LIN {X 0,Y 192.833,Z 984.62,A -85,B 0,C 180,E1 9990.303,E2 9990.303} C_VEL
LIN {X 0,Y 192.693,Z 984.368,A -85,B 0,C 180,E1 9985.841,E2 9985.841} C_VEL
LIN {X 0,Y 192.486,Z 982.897,A -85,B 0,C 180,E1 9980.438,E2 9980.438} C_VEL
LIN {X 0,Y 192.915,Z 979.845,A -85,B 0,C 180,E1 9974.58,E2 9974.58} C_VEL
LIN {X 0,Y 194.824,Z 974.779,A -85,B 0,C 180,E1 9968.005,E2 9968.005} C_VEL
LIN {X 0,Y 198.477,Z 968.183,A -85,B 0,C 180,E1 9961.744,E2 9961.744} C_VEL
LIN {X 0,Y 204.063,Z 959.66,A -85,B 0,C 180,E1 9955.712,E2 9955.712} C_VEL
LIN {X 0,Y 211.597,Z 949.246,A -85,B 0,C 180,E1 9950.02,E2 9950.02} C_VEL
LIN {X 0,Y 220.496,Z 937.345,A -85,B 0,C 180,E1 9944.986,E2 9944.986} C_VEL
LIN {X 0,Y 230.256,Z 924.203,A -85,B 0,C 180,E1 9940.643,E2 9940.643} C_VEL
LIN {X 0,Y 240.936,Z 909.167,A -85,B 0,C 180,E1 9936.792,E2 9936.792} C_VEL
LIN {X 0,Y 251.155,Z 893.767,A -85,B 0,C 180,E1 9933.703,E2 9933.703} C_VEL
LIN {X 0,Y 261.767,Z 876.537,A -85,B 0,C 180,E1 9930.974,E2 9930.974} C_VEL
LIN {X 0,Y 271.504,Z 859.077,A -85,B 0,C 180,E1 9928.793,E2 9928.793} C_VEL
LIN {X 0,Y 280.905,Z 840.055,A -85,B 0,C 180,E1 9926.934,E2 9926.934} C_VEL
LIN {X 0,Y 289.057,Z 821.044,A -85,B 0,C 180,E1 9925.484,E2 9925.484} C_VEL
LIN {X 0,Y 296.643,Z 800.32,A -85,B 0,C 180,E1 9924.267,E2 9924.267} C_VEL
LIN {X 0,Y 302.941,Z 779.468,A -85,B 0,C 180,E1 9923.354,E2 9923.354} C_VEL
LIN {X 0,Y 308.032,Z 757.203,A -85,B 0,C 180,E1 9922.636,E2 9922.636} C_VEL
LIN {X 0,Y 311.388,Z 735.251,A -85,B 0,C 180,E1 9922.089,E2 9922.089} C_VEL
LIN {X 0,Y 327.083,Z 591.178,A -85,B 0,C 180,E1 9919.092,E2 9919.092} C_VEL
LIN {X 0,Y 325.532,Z 586.958,A -85,B 0,C 180,E1 9917.057,E2 9917.057} C_VEL
LIN {X 0,Y 324.558,Z 584.437,A -85,B 0,C 180,E1 9915.363,E2 9915.363} C_VEL
LIN {X 0,Y 323.649,Z 581.615,A -85,B 0,C 180,E1 9912.307,E2 9912.307} C_VEL
LIN {X 0,Y 323.587,Z 581.778,A -85,B 0,C 180,E1 9909.425,E2 9909.425} C_VEL
LIN {X 0,Y 324.621,Z 585.303,A -85,B 0,C 180,E1 9906.011,E2 9906.011} C_VEL
LIN {X 0,Y 326.028,Z 589.355,A -85,B 0,C 180,E1 9903.692,E2 9903.692} C_VEL
LIN {X 0,Y 326.424,Z 590.965,A -85,B 0,C 180,E1 9903.104,E2 9903.104} C_VEL
LIN {X 0,Y 309.523,Z 735.661,A -85,B 0,C 180,E1 9900.051,E2 9900.051} C_VEL
LIN {X 0,Y 305.578,Z 756.66,A -85,B 0,C 180,E1 9899.378,E2 9899.378} C_VEL
LIN {X 0,Y 300.528,Z 776.512,A -85,B 0,C 180,E1 9898.509,E2 9898.509} C_VEL
LIN {X 0,Y 294.236,Z 796.168,A -85,B 0,C 180,E1 9897.379,E2 9897.379} C_VEL
LIN {X 0,Y 287.043,Z 814.874,A -85,B 0,C 180,E1 9896.005,E2 9896.005} C_VEL
LIN {X 0,Y 278.796,Z 832.848,A -85,B 0,C 180,E1 9894.326,E2 9894.326} C_VEL
LIN {X 0,Y 269.408,Z 850.655,A -85,B 0,C 180,E1 9892.227,E2 9892.227} C_VEL
LIN {X 0,Y 259.717,Z 866.928,A -85,B 0,C 180,E1 9889.799,E2 9889.799} C_VEL
LIN {X 0,Y 250.062,Z 881.523,A -85,B 0,C 180,E1 9887.06,E2 9887.06} C_VEL
LIN {X 0,Y 239.647,Z 895.837,A -85,B 0,C 180,E1 9883.636,E2 9883.636} C_VEL
LIN {X 0,Y 229.516,Z 908.579,A -85,B 0,C 180,E1 9879.684,E2 9879.684} C_VEL
LIN {X 0,Y 220.368,Z 919.385,A -85,B 0,C 180,E1 9875.327,E2 9875.327} C_VEL
LIN {X 0,Y 211.892,Z 928.983,A -85,B 0,C 180,E1 9870.24,E2 9870.24} C_VEL
LIN {X 0,Y 205.09,Z 936.539,A -85,B 0,C 180,E1 9864.88,E2 9864.88} C_VEL
LIN {X 0,Y 199.749,Z 942.543,A -85,B 0,C 180,E1 9859.024,E2 9859.024} C_VEL
LIN {X 0,Y 196,Z 946.905,A -85,B 0,C 180,E1 9852.714,E2 9852.714} C_VEL
LIN {X 0,Y 194.012,Z 949.301,A -85,B 0,C 180,E1 9846.704,E2 9846.704} C_VEL
LIN {X 0,Y 193.164,Z 950.247,A -85,B 0,C 180,E1 9840.766,E2 9840.766} C_VEL
LIN {X 0,Y 193.005,Z 949.923,A -85,B 0,C 180,E1 9835.458,E2 9835.458} C_VEL
LIN {X 0,Y 193.369,Z 948.241,A -85,B 0,C 180,E1 9829.765,E2 9829.765} C_VEL
LIN {X 0,Y 194.609,Z 945.069,A -85,B 0,C 180,E1 9823.819,E2 9823.819} C_VEL
LIN {X 0,Y 197.11,Z 940.246,A -85,B 0,C 180,E1 9817.865,E2 9817.865} C_VEL
LIN {X 0,Y 201.137,Z 933.501,A -85,B 0,C 180,E1 9811.988,E2 9811.988} C_VEL
LIN {X 0,Y 206.391,Z 925.353,A -85,B 0,C 180,E1 9806.661,E2 9806.661} C_VEL
LIN {X 0,Y 213.003,Z 915.362,A -85,B 0,C 180,E1 9801.627,E2 9801.627} C_VEL
LIN {X 0,Y 220.514,Z 903.893,A -85,B 0,C 180,E1 9797.129,E2 9797.129} C_VEL
LIN {X 0,Y 228.48,Z 891.228,A -85,B 0,C 180,E1 9793.207,E2 9793.207} C_VEL
LIN {X 0,Y 237.374,Z 876.099,A -85,B 0,C 180,E1 9789.532,E2 9789.532} C_VEL
LIN {X 0,Y 245.848,Z 860.287,A -85,B 0,C 180,E1 9786.507,E2 9786.507} C_VEL
LIN {X 0,Y 253.94,Z 843.552,A -85,B 0,C 180,E1 9783.954,E2 9783.954} C_VEL
LIN {X 0,Y 261.811,Z 825.226,A -85,B 0,C 180,E1 9781.73,E2 9781.73} C_VEL
LIN {X 0,Y 268.975,Z 805.916,A -85,B 0,C 180,E1 9779.874,E2 9779.874} C_VEL
LIN {X 0,Y 274.986,Z 786.777,A -85,B 0,C 180,E1 9778.423,E2 9778.423} C_VEL
LIN {X 0,Y 280.418,Z 765.377,A -85,B 0,C 180,E1 9777.178,E2 9777.178} C_VEL
LIN {X 0,Y 284.657,Z 743.254,A -85,B 0,C 180,E1 9776.242,E2 9776.242} C_VEL
LIN {X 0,Y 287.486,Z 721.546,A -85,B 0,C 180,E1 9775.613,E2 9775.613} C_VEL
LIN {X 0,Y 300.678,Z 576.179,A -85,B 0,C 180,E1 9772.398,E2 9772.398} C_VEL
LIN {X 0,Y 293.024,Z 562.174,A -85,B 0,C 180,E1 9768.58,E2 9768.58} C_VEL
LIN {X 0,Y 286.481,Z 551.351,A -85,B 0,C 180,E1 9764.831,E2 9764.831} C_VEL
LIN {X 0,Y 281.715,Z 543.744,A -85,B 0,C 180,E1 9761.651,E2 9761.651} C_VEL
LIN {X 0,Y 278.454,Z 538.921,A -85,B 0,C 180,E1 9759.197,E2 9759.197} C_VEL
LIN {X 0,Y 275.745,Z 534.842,A -85,B 0,C 180,E1 9756.878,E2 9756.878} C_VEL
LIN {X 0,Y 272.521,Z 530.083,A -85,B 0,C 180,E1 9753.643,E2 9753.643} C_VEL
LIN {X 0,Y 269.339,Z 525.473,A -85,B 0,C 180,E1 9749.587,E2 9749.587} C_VEL
LIN {X 0,Y 266.095,Z 520.826,A -85,B 0,C 180,E1 9742.98,E2 9742.98} C_VEL
LIN {X 0,Y 265.114,Z 519.942,A -85,B 0,C 180,E1 9737.561,E2 9737.561} C_VEL
LIN {X 0,Y 265.642,Z 520.425,A -85,B 0,C 180,E1 9732.389,E2 9732.389} C_VEL
LIN {X 0,Y 266.487,Z 521.324,A -85,B 0,C 180,E1 9729.721,E2 9729.721} C_VEL
LIN {X 0,Y 267.942,Z 523.757,A -85,B 0,C 180,E1 9726.466,E2 9726.466} C_VEL
LIN {X 0,Y 268.633,Z 525.593,A -85,B 0,C 180,E1 9725.108,E2 9725.108} C_VEL
LIN {X 0,Y 269.61,Z 530.896,A -85,B 0,C 180,E1 9723.019,E2 9723.019} C_VEL
LIN {X 0,Y 270.981,Z 536.847,A -85,B 0,C 180,E1 9720.737,E2 9720.737} C_VEL
LIN {X 0,Y 271.921,Z 538.54,A -85,B 0,C 180,E1 9719.631,E2 9719.631} C_VEL
LIN {X 0,Y 276.165,Z 545.02,A -85,B 0,C 180,E1 9715.536,E2 9715.536} C_VEL
LIN {X 0,Y 280.055,Z 550.846,A -85,B 0,C 180,E1 9712.461,E2 9712.461} C_VEL
LIN {X 0,Y 284.859,Z 558.419,A -85,B 0,C 180,E1 9709.177,E2 9709.177} C_VEL
LIN {X 0,Y 291.313,Z 568.942,A -85,B 0,C 180,E1 9705.389,E2 9705.389} C_VEL
LIN {X 0,Y 298.171,Z 581.104,A -85,B 0,C 180,E1 9701.88,E2 9701.88} C_VEL
LIN {X 0,Y 300.746,Z 586.097,A -85,B 0,C 180,E1 9700.666,E2 9700.666} C_VEL
LIN {X 0,Y 286.5,Z 747.246,A -85,B 0,C 180,E1 9697.213,E2 9697.213} C_VEL
LIN {X 0,Y 282.924,Z 769.359,A -85,B 0,C 180,E1 9696.541,E2 9696.541} C_VEL
LIN {X 0,Y 278.126,Z 790.293,A -85,B 0,C 180,E1 9695.696,E2 9695.696} C_VEL
LIN {X 0,Y 272.318,Z 810.598,A -85,B 0,C 180,E1 9694.592,E2 9694.592} C_VEL
LIN {X 0,Y 265.286,Z 830.997,A -85,B 0,C 180,E1 9693.136,E2 9693.136} C_VEL
LIN {X 0,Y 257.466,Z 850.135,A -85,B 0,C 180,E1 9691.368,E2 9691.368} C_VEL
LIN {X 0,Y 249.024,Z 868.363,A -85,B 0,C 180,E1 9689.237,E2 9689.237} C_VEL
LIN {X 0,Y 240.302,Z 885.289,A -85,B 0,C 180,E1 9686.761,E2 9686.761} C_VEL
LIN {X 0,Y 230.867,Z 901.925,A -85,B 0,C 180,E1 9683.669,E2 9683.669} C_VEL
LIN {X 0,Y 221.57,Z 917.018,A -85,B 0,C 180,E1 9680.105,E2 9680.105} C_VEL
LIN {X 0,Y 212.413,Z 931.213,A -85,B 0,C 180,E1 9675.842,E2 9675.842} C_VEL
LIN {X 0,Y 204.126,Z 943.761,A -85,B 0,C 180,E1 9671.03,E2 9671.03} C_VEL
LIN {X 0,Y 197.069,Z 954.627,A -85,B 0,C 180,E1 9665.701,E2 9665.701} C_VEL
LIN {X 0,Y 191.38,Z 963.9,A -85,B 0,C 180,E1 9659.763,E2 9659.763} C_VEL
LIN {X 0,Y 187.435,Z 971.453,A -85,B 0,C 180,E1 9653.436,E2 9653.436} C_VEL
LIN {X 0,Y 185.25,Z 977.221,A -85,B 0,C 180,E1 9646.951,E2 9646.951} C_VEL
LIN {X 0,Y 184.584,Z 980.952,A -85,B 0,C 180,E1 9640.935,E2 9640.935} C_VEL
LIN {X 0,Y 184.709,Z 983.16,A -85,B 0,C 180,E1 9635.123,E2 9635.123} C_VEL
LIN {X 0,Y 184.866,Z 983.888,A -85,B 0,C 180,E1 9630.316,E2 9630.316} C_VEL
LIN {X 0,Y 184.729,Z 983.696,A -85,B 0,C 180,E1 9625.972,E2 9625.972} C_VEL
LIN {X 0,Y 184.506,Z 982.433,A -85,B 0,C 180,E1 9620.651,E2 9620.651} C_VEL
LIN {X 0,Y 184.977,Z 979.342,A -85,B 0,C 180,E1 9614.182,E2 9614.182} C_VEL
LIN {X 0,Y 187.036,Z 974.447,A -85,B 0,C 180,E1 9607.37,E2 9607.37} C_VEL
LIN {X 0,Y 190.947,Z 967.93,A -85,B 0,C 180,E1 9600.866,E2 9600.866} C_VEL
LIN {X 0,Y 196.888,Z 959.58,A -85,B 0,C 180,E1 9594.634,E2 9594.634} C_VEL
LIN {X 0,Y 205.273,Z 948.796,A -85,B 0,C 180,E1 9588.523,E2 9588.523} C_VEL
LIN {X 0,Y 214.698,Z 936.999,A -85,B 0,C 180,E1 9583.417,E2 9583.417} C_VEL
LIN {X 0,Y 225.087,Z 923.789,A -85,B 0,C 180,E1 9578.991,E2 9578.991} C_VEL
LIN {X 0,Y 235.457,Z 909.867,A -85,B 0,C 180,E1 9575.393,E2 9575.393} C_VEL
LIN {X 0,Y 246.713,Z 893.8,A -85,B 0,C 180,E1 9572.123,E2 9572.123} C_VEL
LIN {X 0,Y 257.323,Z 877.334,A -85,B 0,C 180,E1 9569.51,E2 9569.51} C_VEL
LIN {X 0,Y 267.72,Z 859.507,A -85,B 0,C 180,E1 9567.283,E2 9567.283} C_VEL
LIN {X 0,Y 277.372,Z 840.653,A -85,B 0,C 180,E1 9565.46,E2 9565.46} C_VEL
LIN {X 0,Y 286.134,Z 821.067,A -85,B 0,C 180,E1 9563.982,E2 9563.982} C_VEL
LIN {X 0,Y 293.67,Z 801.296,A -85,B 0,C 180,E1 9562.838,E2 9562.838} C_VEL
LIN {X 0,Y 300.384,Z 779.833,A -85,B 0,C 180,E1 9561.914,E2 9561.914} C_VEL
LIN {X 0,Y 305.639,Z 757.703,A -85,B 0,C 180,E1 9561.213,E2 9561.213} C_VEL
LIN {X 0,Y 309.183,Z 735.886,A -85,B 0,C 180,E1 9560.674,E2 9560.674} C_VEL
LIN {X 0,Y 324.902,Z 596.612,A -85,B 0,C 180,E1 9557.784,E2 9557.784} C_VEL
LIN {X 0,Y 323.461,Z 592.436,A -85,B 0,C 180,E1 9555.348,E2 9555.348} C_VEL
LIN {X 0,Y 322.547,Z 589.523,A -85,B 0,C 180,E1 9552.168,E2 9552.168} C_VEL
LIN {X 0,Y 322.489,Z 589.614,A -85,B 0,C 180,E1 9549.638,E2 9549.638} C_VEL
LIN {X 0,Y 323.363,Z 593.042,A -85,B 0,C 180,E1 9546.301,E2 9546.301} C_VEL
LIN {X 0,Y 324.38,Z 596.39,A -85,B 0,C 180,E1 9544.389,E2 9544.389} C_VEL
LIN {X 0,Y 307.554,Z 736.129,A -85,B 0,C 180,E1 9541.49,E2 9541.49} C_VEL
LIN {X 0,Y 303.512,Z 757.009,A -85,B 0,C 180,E1 9540.838,E2 9540.838} C_VEL
LIN {X 0,Y 298.202,Z 777.251,A -85,B 0,C 180,E1 9539.971,E2 9539.971} C_VEL
LIN {X 0,Y 291.469,Z 797.614,A -85,B 0,C 180,E1 9538.82,E2 9538.82} C_VEL
LIN {X 0,Y 284.2,Z 815.824,A -85,B 0,C 180,E1 9537.501,E2 9537.501} C_VEL
LIN {X 0,Y 275.605,Z 833.879,A -85,B 0,C 180,E1 9535.838,E2 9535.838} C_VEL
LIN {X 0,Y 266.445,Z 850.698,A -85,B 0,C 180,E1 9533.892,E2 9533.892} C_VEL
LIN {X 0,Y 256.248,Z 867.217,A -85,B 0,C 180,E1 9531.472,E2 9531.472} C_VEL
LIN {X 0,Y 246.173,Z 881.917,A -85,B 0,C 180,E1 9528.757,E2 9528.757} C_VEL
LIN {X 0,Y 235.124,Z 896.392,A -85,B 0,C 180,E1 9525.31,E2 9525.31} C_VEL
LIN {X 0,Y 225.137,Z 908.385,A -85,B 0,C 180,E1 9521.619,E2 9521.619} C_VEL
LIN {X 0,Y 215.144,Z 919.598,A -85,B 0,C 180,E1 9517.132,E2 9517.132} C_VEL
LIN {X 0,Y 206.072,Z 929.273,A -85,B 0,C 180,E1 9511.998,E2 9511.998} C_VEL
LIN {X 0,Y 198.479,Z 937.134,A -85,B 0,C 180,E1 9506.348,E2 9506.348} C_VEL
LIN {X 0,Y 192.659,Z 943.167,A -85,B 0,C 180,E1 9500.33,E2 9500.33} C_VEL
LIN {X 0,Y 188.407,Z 947.646,A -85,B 0,C 180,E1 9493.611,E2 9493.611} C_VEL
LIN {X 0,Y 186.19,Z 950.04,A -85,B 0,C 180,E1 9487.35,E2 9487.35} C_VEL
LIN {X 0,Y 185.228,Z 950.979,A -85,B 0,C 180,E1 9481.203,E2 9481.203} C_VEL
LIN {X 0,Y 185.035,Z 950.641,A -85,B 0,C 180,E1 9475.522,E2 9475.522} C_VEL
LIN {X 0,Y 185.385,Z 949.048,A -85,B 0,C 180,E1 9469.856,E2 9469.856} C_VEL
LIN {X 0,Y 186.585,Z 946.14,A -85,B 0,C 180,E1 9463.947,E2 9463.947} C_VEL
LIN {X 0,Y 189.209,Z 941.259,A -85,B 0,C 180,E1 9457.585,E2 9457.585} C_VEL
LIN {X 0,Y 193.152,Z 934.985,A -85,B 0,C 180,E1 9451.773,E2 9451.773} C_VEL
LIN {X 0,Y 198.874,Z 926.59,A -85,B 0,C 180,E1 9445.958,E2 9445.958} C_VEL
LIN {X 0,Y 205.756,Z 916.723,A -85,B 0,C 180,E1 9440.766,E2 9440.766} C_VEL
LIN {X 0,Y 213.506,Z 905.467,A -85,B 0,C 180,E1 9436.177,E2 9436.177} C_VEL
LIN {X 0,Y 222.324,Z 892.027,A -85,B 0,C 180,E1 9431.917,E2 9431.917} C_VEL
LIN {X 0,Y 231.494,Z 877.004,A -85,B 0,C 180,E1 9428.222,E2 9428.222} C_VEL
LIN {X 0,Y 240.341,Z 861.098,A -85,B 0,C 180,E1 9425.15,E2 9425.15} C_VEL
LIN {X 0,Y 248.705,Z 844.401,A -85,B 0,C 180,E1 9422.588,E2 9422.588} C_VEL
LIN {X 0,Y 256.822,Z 826.129,A -85,B 0,C 180,E1 9420.363,E2 9420.363} C_VEL
LIN {X 0,Y 263.861,Z 807.884,A -85,B 0,C 180,E1 9418.594,E2 9418.594} C_VEL
LIN {X 0,Y 270.378,Z 787.882,A -85,B 0,C 180,E1 9417.066,E2 9417.066} C_VEL
LIN {X 0,Y 275.951,Z 766.589,A -85,B 0,C 180,E1 9415.828,E2 9415.828} C_VEL
LIN {X 0,Y 280.233,Z 745.122,A -85,B 0,C 180,E1 9414.912,E2 9414.912} C_VEL
LIN {X 0,Y 283.214,Z 723.651,A -85,B 0,C 180,E1 9414.275,E2 9414.275} C_VEL
LIN {X 0,Y 296.636,Z 580.476,A -85,B 0,C 180,E1 9411.135,E2 9411.135} C_VEL
LIN {X 0,Y 289.758,Z 567.709,A -85,B 0,C 180,E1 9407.519,E2 9407.519} C_VEL
LIN {X 0,Y 283.334,Z 556.902,A -85,B 0,C 180,E1 9403.623,E2 9403.623} C_VEL
LIN {X 0,Y 278.597,Z 549.234,A -85,B 0,C 180,E1 9400.242,E2 9400.242} C_VEL
LIN {X 0,Y 274.037,Z 542.29,A -85,B 0,C 180,E1 9396.364,E2 9396.364} C_VEL
LIN {X 0,Y 271.016,Z 537.705,A -85,B 0,C 180,E1 9393.221,E2 9393.221} C_VEL
LIN {X 0,Y 267.959,Z 533.166,A -85,B 0,C 180,E1 9389.168,E2 9389.168} C_VEL
LIN {X 0,Y 264.982,Z 528.733,A -85,B 0,C 180,E1 9382.871,E2 9382.871} C_VEL
LIN {X 0,Y 264.034,Z 527.866,A -85,B 0,C 180,E1 9377.381,E2 9377.381} C_VEL
LIN {X 0,Y 264.615,Z 528.399,A -85,B 0,C 180,E1 9372.217,E2 9372.217} C_VEL
LIN {X 0,Y 265.391,Z 529.314,A -85,B 0,C 180,E1 9369.762,E2 9369.762} C_VEL
LIN {X 0,Y 268.904,Z 534.267,A -85,B 0,C 180,E1 9363.305,E2 9363.305} C_VEL
LIN {X 0,Y 271.921,Z 538.54,A -85,B 0,C 180,E1 9359.631,E2 9359.631} C_VEL
LIN {X 0,Y 273.084,Z 540.822,A -85,B 0,C 180,E1 9358.351,E2 9358.351} C_VEL
LIN {X 0,Y 274.504,Z 546.424,A -85,B 0,C 180,E1 9356.636,E2 9356.636} C_VEL
LIN {X 0,Y 276.478,Z 554.666,A -85,B 0,C 180,E1 9354.425,E2 9354.425} C_VEL
LIN {X 0,Y 277.625,Z 557.294,A -85,B 0,C 180,E1 9353.422,E2 9353.422} C_VEL
LIN {X 0,Y 282.668,Z 565.44,A -85,B 0,C 180,E1 9349.814,E2 9349.814} C_VEL
LIN {X 0,Y 288.966,Z 575.986,A -85,B 0,C 180,E1 9345.984,E2 9345.984} C_VEL
LIN {X 0,Y 295.773,Z 588.381,A -85,B 0,C 180,E1 9342.389,E2 9342.389} C_VEL
LIN {X 0,Y 296.668,Z 590.18,A -85,B 0,C 180,E1 9341.944,E2 9341.944} C_VEL
LIN {X 0,Y 282.411,Z 747.03,A -85,B 0,C 180,E1 9338.602,E2 9338.602} C_VEL
LIN {X 0,Y 278.737,Z 769.213,A -85,B 0,C 180,E1 9337.934,E2 9337.934} C_VEL
LIN {X 0,Y 273.812,Z 790.175,A -85,B 0,C 180,E1 9337.098,E2 9337.098} C_VEL
LIN {X 0,Y 267.699,Z 810.918,A -85,B 0,C 180,E1 9335.977,E2 9335.977} C_VEL
LIN {X 0,Y 260.565,Z 831.016,A -85,B 0,C 180,E1 9334.547,E2 9334.547} C_VEL
LIN {X 0,Y 252.454,Z 850.268,A -85,B 0,C 180,E1 9332.773,E2 9332.773} C_VEL
LIN {X 0,Y 243.777,Z 868.376,A -85,B 0,C 180,E1 9330.649,E2 9330.649} C_VEL
LIN {X 0,Y 234.454,Z 885.785,A -85,B 0,C 180,E1 9328.073,E2 9328.073} C_VEL
LIN {X 0,Y 224.73,Z 902.341,A -85,B 0,C 180,E1 9324.956,E2 9324.956} C_VEL
LIN {X 0,Y 215.12,Z 917.318,A -85,B 0,C 180,E1 9321.345,E2 9321.345} C_VEL
LIN {X 0,Y 205.926,Z 930.916,A -85,B 0,C 180,E1 9317.159,E2 9317.159} C_VEL
LIN {X 0,Y 197.333,Z 943.293,A -85,B 0,C 180,E1 9312.29,E2 9312.29} C_VEL
LIN {X 0,Y 189.965,Z 954.037,A -85,B 0,C 180,E1 9306.868,E2 9306.868} C_VEL
LIN {X 0,Y 183.925,Z 963.302,A -85,B 0,C 180,E1 9300.737,E2 9300.737} C_VEL
LIN {X 0,Y 179.77,Z 970.689,A -85,B 0,C 180,E1 9294.311,E2 9294.311} C_VEL
LIN {X 0,Y 177.417,Z 976.359,A -85,B 0,C 180,E1 9287.724,E2 9287.724} C_VEL
LIN {X 0,Y 176.622,Z 980.126,A -85,B 0,C 180,E1 9281.435,E2 9281.435} C_VEL
LIN {X 0,Y 176.731,Z 982.41,A -85,B 0,C 180,E1 9275.312,E2 9275.312} C_VEL
LIN {X 0,Y 176.899,Z 983.157,A -85,B 0,C 180,E1 9270.331,E2 9270.331} C_VEL
LIN {X 0,Y 176.746,Z 982.982,A -85,B 0,C 180,E1 9265.79,E2 9265.79} C_VEL
LIN {X 0,Y 176.522,Z 981.732,A -85,B 0,C 180,E1 9260.224,E2 9260.224} C_VEL
LIN {X 0,Y 177.069,Z 978.772,A -85,B 0,C 180,E1 9253.608,E2 9253.608} C_VEL
LIN {X 0,Y 179.27,Z 974.121,A -85,B 0,C 180,E1 9246.68,E2 9246.68} C_VEL
LIN {X 0,Y 183.465,Z 967.693,A -85,B 0,C 180,E1 9239.917,E2 9239.917} C_VEL
LIN {X 0,Y 189.789,Z 959.502,A -85,B 0,C 180,E1 9233.474,E2 9233.474} C_VEL
LIN {X 0,Y 198.199,Z 949.467,A -85,B 0,C 180,E1 9227.479,E2 9227.479} C_VEL
LIN {X 0,Y 208.007,Z 937.998,A -85,B 0,C 180,E1 9222.258,E2 9222.258} C_VEL
LIN {X 0,Y 218.763,Z 924.999,A -85,B 0,C 180,E1 9217.761,E2 9217.761} C_VEL
LIN {X 0,Y 230.132,Z 910.653,A -85,B 0,C 180,E1 9213.93,E2 9213.93} C_VEL
LIN {X 0,Y 242.116,Z 894.38,A -85,B 0,C 180,E1 9210.58,E2 9210.58} C_VEL
LIN {X 0,Y 253.061,Z 878.242,A -85,B 0,C 180,E1 9208,E2 9208} C_VEL
LIN {X 0,Y 264.552,Z 859.227,A -85,B 0,C 180,E1 9205.652,E2 9205.652} C_VEL
LIN {X 0,Y 274.44,Z 840.62,A -85,B 0,C 180,E1 9203.886,E2 9203.886} C_VEL
LIN {X 0,Y 283.832,Z 820.224,A -85,B 0,C 180,E1 9202.391,E2 9202.391} C_VEL
LIN {X 0,Y 291.786,Z 799.829,A -85,B 0,C 180,E1 9201.258,E2 9201.258} C_VEL
LIN {X 0,Y 298.408,Z 779.132,A -85,B 0,C 180,E1 9200.407,E2 9200.407} C_VEL
LIN {X 0,Y 303.791,Z 756.859,A -85,B 0,C 180,E1 9199.728,E2 9199.728} C_VEL
LIN {X 0,Y 307.441,Z 734.943,A -85,B 0,C 180,E1 9199.203,E2 9199.203} C_VEL
LIN {X 0,Y 322.953,Z 602.452,A -85,B 0,C 180,E1 9196.502,E2 9196.502} C_VEL
LIN {X 0,Y 322.097,Z 599.9,A -85,B 0,C 180,E1 9194.746,E2 9194.746} C_VEL
LIN {X 0,Y 321.441,Z 597.431,A -85,B 0,C 180,E1 9192.028,E2 9192.028} C_VEL
LIN {X 0,Y 321.388,Z 597.633,A -85,B 0,C 180,E1 9189.671,E2 9189.671} C_VEL
LIN {X 0,Y 322.111,Z 600.78,A -85,B 0,C 180,E1 9186.595,E2 9186.595} C_VEL
LIN {X 0,Y 322.487,Z 602.369,A -85,B 0,C 180,E1 9185.68,E2 9185.68} C_VEL
LIN {X 0,Y 305.848,Z 736.59,A -85,B 0,C 180,E1 9182.949,E2 9182.949} C_VEL
LIN {X 0,Y 301.647,Z 757.664,A -85,B 0,C 180,E1 9182.308,E2 9182.308} C_VEL
LIN {X 0,Y 296.367,Z 777.386,A -85,B 0,C 180,E1 9181.49,E2 9181.49} C_VEL
LIN {X 0,Y 289.582,Z 797.446,A -85,B 0,C 180,E1 9180.395,E2 9180.395} C_VEL
LIN {X 0,Y 281.646,Z 816.695,A -85,B 0,C 180,E1 9179.036,E2 9179.036} C_VEL
LIN {X 0,Y 272.714,Z 834.906,A -85,B 0,C 180,E1 9177.395,E2 9177.395} C_VEL
LIN {X 0,Y 262.923,Z 852.151,A -85,B 0,C 180,E1 9175.419,E2 9175.419} C_VEL
LIN {X 0,Y 251.862,Z 869.301,A -85,B 0,C 180,E1 9172.908,E2 9172.908} C_VEL
LIN {X 0,Y 241.026,Z 884.238,A -85,B 0,C 180,E1 9170.1,E2 9170.1} C_VEL
LIN {X 0,Y 230.033,Z 897.994,A -85,B 0,C 180,E1 9166.784,E2 9166.784} C_VEL
LIN {X 0,Y 219.142,Z 910.356,A -85,B 0,C 180,E1 9162.89,E2 9162.89} C_VEL
LIN {X 0,Y 209.337,Z 920.709,A -85,B 0,C 180,E1 9158.631,E2 9158.631} C_VEL
LIN {X 0,Y 199.919,Z 930.11,A -85,B 0,C 180,E1 9153.521,E2 9153.521} C_VEL
LIN {X 0,Y 192.016,Z 937.749,A -85,B 0,C 180,E1 9147.917,E2 9147.917} C_VEL
LIN {X 0,Y 185.674,Z 943.797,A -85,B 0,C 180,E1 9141.736,E2 9141.736} C_VEL
LIN {X 0,Y 181.057,Z 948.186,A -85,B 0,C 180,E1 9134.969,E2 9134.969} C_VEL
LIN {X 0,Y 178.469,Z 950.7,A -85,B 0,C 180,E1 9128.339,E2 9128.339} C_VEL
LIN {X 0,Y 177.299,Z 951.716,A -85,B 0,C 180,E1 9121.618,E2 9121.618} C_VEL
LIN {X 0,Y 177.063,Z 951.379,A -85,B 0,C 180,E1 9115.765,E2 9115.765} C_VEL
LIN {X 0,Y 177.424,Z 949.776,A -85,B 0,C 180,E1 9109.755,E2 9109.755} C_VEL
LIN {X 0,Y 178.698,Z 946.872,A -85,B 0,C 180,E1 9103.584,E2 9103.584} C_VEL
LIN {X 0,Y 181.493,Z 941.99,A -85,B 0,C 180,E1 9096.954,E2 9096.954} C_VEL
LIN {X 0,Y 185.678,Z 935.723,A -85,B 0,C 180,E1 9090.919,E2 9090.919} C_VEL
LIN {X 0,Y 191.734,Z 927.322,A -85,B 0,C 180,E1 9084.902,E2 9084.902} C_VEL
LIN {X 0,Y 198.967,Z 917.472,A -85,B 0,C 180,E1 9079.571,E2 9079.571} C_VEL
LIN {X 0,Y 207.085,Z 906.228,A -85,B 0,C 180,E1 9074.881,E2 9074.881} C_VEL
LIN {X 0,Y 216.285,Z 892.799,A -85,B 0,C 180,E1 9070.553,E2 9070.553} C_VEL
LIN {X 0,Y 225.292,Z 878.607,A -85,B 0,C 180,E1 9067.006,E2 9067.006} C_VEL
LIN {X 0,Y 234.35,Z 863.02,A -85,B 0,C 180,E1 9063.926,E2 9063.926} C_VEL
LIN {X 0,Y 243.288,Z 845.903,A -85,B 0,C 180,E1 9061.255,E2 9061.255} C_VEL
LIN {X 0,Y 251.64,Z 827.8,A -85,B 0,C 180,E1 9059.028,E2 9059.028} C_VEL
LIN {X 0,Y 258.877,Z 809.786,A -85,B 0,C 180,E1 9057.263,E2 9057.263} C_VEL
LIN {X 0,Y 265.541,Z 790.017,A -85,B 0,C 180,E1 9055.744,E2 9055.744} C_VEL
LIN {X 0,Y 271.09,Z 769.788,A -85,B 0,C 180,E1 9054.546,E2 9054.546} C_VEL
LIN {X 0,Y 275.682,Z 748.23,A -85,B 0,C 180,E1 9053.594,E2 9053.594} C_VEL
LIN {X 0,Y 279.065,Z 725.551,A -85,B 0,C 180,E1 9052.9,E2 9052.9} C_VEL
LIN {X 0,Y 292.657,Z 584.756,A -85,B 0,C 180,E1 9049.823,E2 9049.823} C_VEL
LIN {X 0,Y 286.599,Z 573.391,A -85,B 0,C 180,E1 9046.451,E2 9046.451} C_VEL
LIN {X 0,Y 280.78,Z 563.239,A -85,B 0,C 180,E1 9042.717,E2 9042.717} C_VEL
LIN {X 0,Y 275.847,Z 555.059,A -85,B 0,C 180,E1 9038.968,E2 9038.968} C_VEL
LIN {X 0,Y 272.238,Z 549.579,A -85,B 0,C 180,E1 9035.731,E2 9035.731} C_VEL
LIN {X 0,Y 269.525,Z 545.326,A -85,B 0,C 180,E1 9032.795,E2 9032.795} C_VEL
LIN {X 0,Y 266.706,Z 540.984,A -85,B 0,C 180,E1 9028.922,E2 9028.922} C_VEL
LIN {X 0,Y 263.793,Z 536.569,A -85,B 0,C 180,E1 9022.509,E2 9022.509} C_VEL
LIN {X 0,Y 262.951,Z 535.78,A -85,B 0,C 180,E1 9017.026,E2 9017.026} C_VEL
LIN {X 0,Y 263.655,Z 536.42,A -85,B 0,C 180,E1 9011.818,E2 9011.818} C_VEL
LIN {X 0,Y 264.294,Z 537.302,A -85,B 0,C 180,E1 9009.802,E2 9009.802} C_VEL
LIN {X 0,Y 267.64,Z 542.148,A -85,B 0,C 180,E1 9003.535,E2 9003.535} C_VEL
LIN {X 0,Y 271.021,Z 547.224,A -85,B 0,C 180,E1 8999.366,E2 8999.366} C_VEL
LIN {X 0,Y 274.451,Z 552.464,A -85,B 0,C 180,E1 8996.031,E2 8996.031} C_VEL
LIN {X 0,Y 277.625,Z 557.294,A -85,B 0,C 180,E1 8993.422,E2 8993.422} C_VEL
LIN {X 0,Y 279.241,Z 561.173,A -85,B 0,C 180,E1 8992.082,E2 8992.082} C_VEL
LIN {X 0,Y 281.518,Z 570.097,A -85,B 0,C 180,E1 8990.083,E2 8990.083} C_VEL
LIN {X 0,Y 283.661,Z 577.43,A -85,B 0,C 180,E1 8988.408,E2 8988.408} C_VEL
LIN {X 0,Y 284.501,Z 579.252,A -85,B 0,C 180,E1 8987.863,E2 8987.863} C_VEL
LIN {X 0,Y 290.309,Z 589.84,A -85,B 0,C 180,E1 8984.52,E2 8984.52} C_VEL
LIN {X 0,Y 292.711,Z 594.573,A -85,B 0,C 180,E1 8983.25,E2 8983.25} C_VEL
LIN {X 0,Y 278.461,Z 746.627,A -85,B 0,C 180,E1 8980.03,E2 8980.03} C_VEL
LIN {X 0,Y 274.717,Z 768.754,A -85,B 0,C 180,E1 8979.371,E2 8979.371} C_VEL
LIN {X 0,Y 269.664,Z 789.808,A -85,B 0,C 180,E1 8978.545,E2 8978.545} C_VEL
LIN {X 0,Y 263.186,Z 811.189,A -85,B 0,C 180,E1 8977.402,E2 8977.402} C_VEL
LIN {X 0,Y 256.072,Z 830.722,A -85,B 0,C 180,E1 8976.026,E2 8976.026} C_VEL
LIN {X 0,Y 247.599,Z 850.33,A -85,B 0,C 180,E1 8974.235,E2 8974.235} C_VEL
LIN {X 0,Y 238.683,Z 868.367,A -85,B 0,C 180,E1 8972.123,E2 8972.123} C_VEL
LIN {X 0,Y 228.735,Z 886.28,A -85,B 0,C 180,E1 8969.452,E2 8969.452} C_VEL
LIN {X 0,Y 219.331,Z 901.723,A -85,B 0,C 180,E1 8966.524,E2 8966.524} C_VEL
LIN {X 0,Y 209.371,Z 916.662,A -85,B 0,C 180,E1 8962.901,E2 8962.901} C_VEL
LIN {X 0,Y 199.69,Z 930.383,A -85,B 0,C 180,E1 8958.63,E2 8958.63} C_VEL
LIN {X 0,Y 190.384,Z 943.158,A -85,B 0,C 180,E1 8953.478,E2 8953.478} C_VEL
LIN {X 0,Y 182.87,Z 953.537,A -85,B 0,C 180,E1 8948.065,E2 8948.065} C_VEL
LIN {X 0,Y 176.526,Z 962.679,A -85,B 0,C 180,E1 8941.794,E2 8941.794} C_VEL
LIN {X 0,Y 172.066,Z 970.053,A -85,B 0,C 180,E1 8935.107,E2 8935.107} C_VEL
LIN {X 0,Y 169.524,Z 975.708,A -85,B 0,C 180,E1 8928.223,E2 8928.223} C_VEL
LIN {X 0,Y 168.648,Z 979.466,A -85,B 0,C 180,E1 8921.636,E2 8921.636} C_VEL
LIN {X 0,Y 168.757,Z 981.672,A -85,B 0,C 180,E1 8915.447,E2 8915.447} C_VEL
LIN {X 0,Y 168.932,Z 982.423,A -85,B 0,C 180,E1 8910.346,E2 8910.346} C_VEL
LIN {X 0,Y 168.763,Z 982.27,A -85,B 0,C 180,E1 8905.59,E2 8905.59} C_VEL
LIN {X 0,Y 168.543,Z 981.099,A -85,B 0,C 180,E1 8899.983,E2 8899.983} C_VEL
LIN {X 0,Y 169.212,Z 978.119,A -85,B 0,C 180,E1 8892.824,E2 8892.824} C_VEL
LIN {X 0,Y 171.694,Z 973.524,A -85,B 0,C 180,E1 8885.586,E2 8885.586} C_VEL
LIN {X 0,Y 176.584,Z 966.792,A -85,B 0,C 180,E1 8878.234,E2 8878.234} C_VEL
LIN {X 0,Y 183.535,Z 958.594,A -85,B 0,C 180,E1 8871.617,E2 8871.617} C_VEL
LIN {X 0,Y 192.615,Z 948.54,A -85,B 0,C 180,E1 8865.521,E2 8865.521} C_VEL
LIN {X 0,Y 203.07,Z 937.065,A -85,B 0,C 180,E1 8860.266,E2 8860.266} C_VEL
LIN {X 0,Y 214.435,Z 924.102,A -85,B 0,C 180,E1 8855.787,E2 8855.787} C_VEL
LIN {X 0,Y 226.338,Z 909.753,A -85,B 0,C 180,E1 8852,E2 8852} C_VEL
LIN {X 0,Y 238.437,Z 894.022,A -85,B 0,C 180,E1 8848.801,E2 8848.801} C_VEL
LIN {X 0,Y 249.945,Z 877.707,A -85,B 0,C 180,E1 8846.237,E2 8846.237} C_VEL
LIN {X 0,Y 261.116,Z 859.855,A -85,B 0,C 180,E1 8844.075,E2 8844.075} C_VEL
LIN {X 0,Y 271.314,Z 841.483,A -85,B 0,C 180,E1 8842.349,E2 8842.349} C_VEL
LIN {X 0,Y 280.918,Z 821.522,A -85,B 0,C 180,E1 8840.901,E2 8840.901} C_VEL
LIN {X 0,Y 289.035,Z 801.68,A -85,B 0,C 180,E1 8839.809,E2 8839.809} C_VEL
LIN {X 0,Y 295.99,Z 780.791,A -85,B 0,C 180,E1 8838.96,E2 8838.96} C_VEL
LIN {X 0,Y 301.537,Z 759.265,A -85,B 0,C 180,E1 8838.309,E2 8838.309} C_VEL
LIN {X 0,Y 305.682,Z 736.194,A -85,B 0,C 180,E1 8837.759,E2 8837.759} C_VEL
LIN {X 0,Y 321.172,Z 608.612,A -85,B 0,C 180,E1 8835.208,E2 8835.208} C_VEL
LIN {X 0,Y 320.337,Z 605.339,A -85,B 0,C 180,E1 8831.888,E2 8831.888} C_VEL
LIN {X 0,Y 320.29,Z 605.469,A -85,B 0,C 180,E1 8829.886,E2 8829.886} C_VEL
LIN {X 0,Y 320.833,Z 608.382,A -85,B 0,C 180,E1 8826.986,E2 8826.986} C_VEL
LIN {X 0,Y 304.394,Z 737.285,A -85,B 0,C 180,E1 8824.42,E2 8824.42} C_VEL
LIN {X 0,Y 300.107,Z 758.295,A -85,B 0,C 180,E1 8823.8,E2 8823.8} C_VEL
LIN {X 0,Y 294.606,Z 778.207,A -85,B 0,C 180,E1 8822.998,E2 8822.998} C_VEL
LIN {X 0,Y 287.593,Z 798.265,A -85,B 0,C 180,E1 8821.932,E2 8821.932} C_VEL
LIN {X 0,Y 279.456,Z 817.462,A -85,B 0,C 180,E1 8820.614,E2 8820.614} C_VEL
LIN {X 0,Y 270.468,Z 835.208,A -85,B 0,C 180,E1 8819.059,E2 8819.059} C_VEL
LIN {X 0,Y 260.264,Z 852.648,A -85,B 0,C 180,E1 8817.114,E2 8817.114} C_VEL
LIN {X 0,Y 248.992,Z 869.552,A -85,B 0,C 180,E1 8814.7,E2 8814.7} C_VEL
LIN {X 0,Y 238.071,Z 884.128,A -85,B 0,C 180,E1 8812.033,E2 8812.033} C_VEL
LIN {X 0,Y 226.325,Z 898.23,A -85,B 0,C 180,E1 8808.703,E2 8808.703} C_VEL
LIN {X 0,Y 214.537,Z 911.015,A -85,B 0,C 180,E1 8804.71,E2 8804.71} C_VEL
LIN {X 0,Y 203.649,Z 921.87,A -85,B 0,C 180,E1 8800.197,E2 8800.197} C_VEL
LIN {X 0,Y 193.597,Z 931.287,A -85,B 0,C 180,E1 8794.943,E2 8794.943} C_VEL
LIN {X 0,Y 185.111,Z 938.88,A -85,B 0,C 180,E1 8789.126,E2 8789.126} C_VEL
LIN {X 0,Y 178.353,Z 944.821,A -85,B 0,C 180,E1 8782.737,E2 8782.737} C_VEL
LIN {X 0,Y 173.373,Z 949.161,A -85,B 0,C 180,E1 8775.641,E2 8775.641} C_VEL
LIN {X 0,Y 170.612,Z 951.54,A -85,B 0,C 180,E1 8768.789,E2 8768.789} C_VEL
LIN {X 0,Y 169.337,Z 952.456,A -85,B 0,C 180,E1 8761.693,E2 8761.693} C_VEL
LIN {X 0,Y 169.098,Z 952.065,A -85,B 0,C 180,E1 8755.563,E2 8755.563} C_VEL
LIN {X 0,Y 169.512,Z 950.367,A -85,B 0,C 180,E1 8749.279,E2 8749.279} C_VEL
LIN {X 0,Y 171.035,Z 947.153,A -85,B 0,C 180,E1 8742.484,E2 8742.484} C_VEL
LIN {X 0,Y 174.199,Z 942.156,A -85,B 0,C 180,E1 8735.592,E2 8735.592} C_VEL
LIN {X 0,Y 179.102,Z 935.352,A -85,B 0,C 180,E1 8729.034,E2 8729.034} C_VEL
LIN {X 0,Y 185.382,Z 927.124,A -85,B 0,C 180,E1 8723.179,E2 8723.179} C_VEL
LIN {X 0,Y 193.154,Z 917.044,A -85,B 0,C 180,E1 8717.74,E2 8717.74} C_VEL
LIN {X 0,Y 201.816,Z 905.507,A -85,B 0,C 180,E1 8712.979,E2 8712.979} C_VEL
LIN {X 0,Y 210.931,Z 892.698,A -85,B 0,C 180,E1 8708.879,E2 8708.879} C_VEL
LIN {X 0,Y 220.337,Z 878.408,A -85,B 0,C 180,E1 8705.319,E2 8705.319} C_VEL
LIN {X 0,Y 229.753,Z 862.643,A -85,B 0,C 180,E1 8702.243,E2 8702.243} C_VEL
LIN {X 0,Y 238.509,Z 846.318,A -85,B 0,C 180,E1 8699.722,E2 8699.722} C_VEL
LIN {X 0,Y 247.291,Z 827.786,A -85,B 0,C 180,E1 8697.465,E2 8697.465} C_VEL
LIN {X 0,Y 254.867,Z 809.292,A -85,B 0,C 180,E1 8695.686,E2 8695.686} C_VEL
LIN {X 0,Y 261.61,Z 789.74,A -85,B 0,C 180,E1 8694.21,E2 8694.21} C_VEL
LIN {X 0,Y 267.211,Z 769.663,A -85,B 0,C 180,E1 8693.047,E2 8693.047} C_VEL
LIN {X 0,Y 271.844,Z 748.301,A -85,B 0,C 180,E1 8692.122,E2 8692.122} C_VEL
LIN {X 0,Y 275.282,Z 725.694,A -85,B 0,C 180,E1 8691.442,E2 8691.442} C_VEL
LIN {X 0,Y 288.808,Z 589.059,A -85,B 0,C 180,E1 8688.475,E2 8688.475} C_VEL
LIN {X 0,Y 283.775,Z 579.461,A -85,B 0,C 180,E1 8685.506,E2 8685.506} C_VEL
LIN {X 0,Y 278.038,Z 569.141,A -85,B 0,C 180,E1 8681.623,E2 8681.623} C_VEL
LIN {X 0,Y 273.401,Z 561.555,A -85,B 0,C 180,E1 8677.909,E2 8677.909} C_VEL
LIN {X 0,Y 270.571,Z 557.02,A -85,B 0,C 180,E1 8675.204,E2 8675.204} C_VEL
LIN {X 0,Y 268.049,Z 552.946,A -85,B 0,C 180,E1 8672.363,E2 8672.363} C_VEL
LIN {X 0,Y 265.403,Z 548.74,A -85,B 0,C 180,E1 8668.585,E2 8668.585} C_VEL
LIN {X 0,Y 262.663,Z 544.456,A -85,B 0,C 180,E1 8662.322,E2 8662.322} C_VEL
LIN {X 0,Y 261.877,Z 543.702,A -85,B 0,C 180,E1 8656.869,E2 8656.869} C_VEL
LIN {X 0,Y 262.707,Z 544.447,A -85,B 0,C 180,E1 8651.415,E2 8651.415} C_VEL
LIN {X 0,Y 263.787,Z 546.473,A -85,B 0,C 180,E1 8648.282,E2 8648.282} C_VEL
LIN {X 0,Y 266.306,Z 549.883,A -85,B 0,C 180,E1 8643.876,E2 8643.876} C_VEL
LIN {X 0,Y 269.516,Z 554.832,A -85,B 0,C 180,E1 8639.788,E2 8639.788} C_VEL
LIN {X 0,Y 272.864,Z 560.1,A -85,B 0,C 180,E1 8636.429,E2 8636.429} C_VEL
LIN {X 0,Y 276.79,Z 566.26,A -85,B 0,C 180,E1 8633.154,E2 8633.154} C_VEL
LIN {X 0,Y 281.961,Z 574.853,A -85,B 0,C 180,E1 8629.478,E2 8629.478} C_VEL
LIN {X 0,Y 284.501,Z 579.252,A -85,B 0,C 180,E1 8627.863,E2 8627.863} C_VEL
LIN {X 0,Y 285.595,Z 582.684,A -85,B 0,C 180,E1 8627.105,E2 8627.105} C_VEL
LIN {X 0,Y 287.436,Z 595.248,A -85,B 0,C 180,E1 8625.427,E2 8625.427} C_VEL
LIN {X 0,Y 288.315,Z 597.695,A -85,B 0,C 180,E1 8624.887,E2 8624.887} C_VEL
LIN {X 0,Y 288.831,Z 599.021,A -85,B 0,C 180,E1 8624.583,E2 8624.583} C_VEL
LIN {X 0,Y 274.676,Z 746.227,A -85,B 0,C 180,E1 8621.496,E2 8621.496} C_VEL
LIN {X 0,Y 270.847,Z 768.418,A -85,B 0,C 180,E1 8620.845,E2 8620.845} C_VEL
LIN {X 0,Y 265.693,Z 789.434,A -85,B 0,C 180,E1 8620.037,E2 8620.037} C_VEL
LIN {X 0,Y 259.052,Z 810.849,A -85,B 0,C 180,E1 8618.912,E2 8618.912} C_VEL
LIN {X 0,Y 251.591,Z 830.76,A -85,B 0,C 180,E1 8617.525,E2 8617.525} C_VEL
LIN {X 0,Y 242.908,Z 850.307,A -85,B 0,C 180,E1 8615.755,E2 8615.755} C_VEL
LIN {X 0,Y 233.752,Z 868.252,A -85,B 0,C 180,E1 8613.661,E2 8613.661} C_VEL
LIN {X 0,Y 223.667,Z 885.845,A -85,B 0,C 180,E1 8611.046,E2 8611.046} C_VEL
LIN {X 0,Y 213.486,Z 901.961,A -85,B 0,C 180,E1 8607.971,E2 8607.971} C_VEL
LIN {X 0,Y 203.164,Z 916.894,A -85,B 0,C 180,E1 8604.303,E2 8604.303} C_VEL
LIN {X 0,Y 193.191,Z 930.369,A -85,B 0,C 180,E1 8600.001,E2 8600.001} C_VEL
LIN {X 0,Y 183.42,Z 943.114,A -85,B 0,C 180,E1 8594.692,E2 8594.692} C_VEL
LIN {X 0,Y 175.271,Z 953.747,A -85,B 0,C 180,E1 8588.874,E2 8588.874} C_VEL
LIN {X 0,Y 168.617,Z 962.909,A -85,B 0,C 180,E1 8582.262,E2 8582.262} C_VEL
LIN {X 0,Y 164.034,Z 970.061,A -85,B 0,C 180,E1 8575.265,E2 8575.265} C_VEL
LIN {X 0,Y 161.386,Z 975.715,A -85,B 0,C 180,E1 8567.68,E2 8567.68} C_VEL
LIN {X 0,Y 160.639,Z 979.297,A -85,B 0,C 180,E1 8560.769,E2 8560.769} C_VEL
LIN {X 0,Y 160.818,Z 981.109,A -85,B 0,C 180,E1 8554.643,E2 8554.643} C_VEL
LIN {X 0,Y 160.962,Z 981.714,A -85,B 0,C 180,E1 8549.652,E2 8549.652} C_VEL
LIN {X 0,Y 160.748,Z 981.473,A -85,B 0,C 180,E1 8544.654,E2 8544.654} C_VEL
LIN {X 0,Y 160.598,Z 980.054,A -85,B 0,C 180,E1 8538.152,E2 8538.152} C_VEL
LIN {X 0,Y 161.758,Z 976.72,A -85,B 0,C 180,E1 8530.51,E2 8530.51} C_VEL
LIN {X 0,Y 165.392,Z 971.238,A -85,B 0,C 180,E1 8522.267,E2 8522.267} C_VEL
LIN {X 0,Y 171.138,Z 964.518,A -85,B 0,C 180,E1 8515.081,E2 8515.081} C_VEL
LIN {X 0,Y 179.624,Z 955.533,A -85,B 0,C 180,E1 8508.1,E2 8508.1} C_VEL
LIN {X 0,Y 189.896,Z 944.945,A -85,B 0,C 180,E1 8502.075,E2 8502.075} C_VEL
LIN {X 0,Y 201.428,Z 932.921,A -85,B 0,C 180,E1 8496.961,E2 8496.961} C_VEL
LIN {X 0,Y 213.733,Z 919.486,A -85,B 0,C 180,E1 8492.656,E2 8492.656} C_VEL
LIN {X 0,Y 226.438,Z 904.617,A -85,B 0,C 180,E1 8489.053,E2 8489.053} C_VEL
LIN {X 0,Y 238.838,Z 888.684,A -85,B 0,C 180,E1 8486.123,E2 8486.123} C_VEL
LIN {X 0,Y 250.618,Z 871.935,A -85,B 0,C 180,E1 8483.762,E2 8483.762} C_VEL
LIN {X 0,Y 262.119,Z 853.601,A -85,B 0,C 180,E1 8481.763,E2 8481.763} C_VEL
LIN {X 0,Y 272.219,Z 835.307,A -85,B 0,C 180,E1 8480.225,E2 8480.225} C_VEL
LIN {X 0,Y 281.238,Z 816.178,A -85,B 0,C 180,E1 8478.989,E2 8478.989} C_VEL
LIN {X 0,Y 289.112,Z 796.389,A -85,B 0,C 180,E1 8478.02,E2 8478.02} C_VEL
LIN {X 0,Y 296.112,Z 774.815,A -85,B 0,C 180,E1 8477.242,E2 8477.242} C_VEL
LIN {X 0,Y 301.498,Z 752.99,A -85,B 0,C 180,E1 8476.644,E2 8476.644} C_VEL
LIN {X 0,Y 305.263,Z 730.155,A -85,B 0,C 180,E1 8476.146,E2 8476.146} C_VEL
LIN {X 0,Y 319.593,Z 615.147,A -85,B 0,C 180,E1 8473.893,E2 8473.893} C_VEL
LIN {X 0,Y 319.235,Z 613.248,A -85,B 0,C 180,E1 8471.746,E2 8471.746} C_VEL
LIN {X 0,Y 319.189,Z 613.486,A -85,B 0,C 180,E1 8469.92,E2 8469.92} C_VEL
LIN {X 0,Y 319.342,Z 615.128,A -85,B 0,C 180,E1 8468.294,E2 8468.294} C_VEL
LIN {X 0,Y 303.282,Z 737.768,A -85,B 0,C 180,E1 8465.913,E2 8465.913} C_VEL
LIN {X 0,Y 298.867,Z 758.826,A -85,B 0,C 180,E1 8465.313,E2 8465.313} C_VEL
LIN {X 0,Y 293.355,Z 778.295,A -85,B 0,C 180,E1 8464.558,E2 8464.558} C_VEL
LIN {X 0,Y 285.963,Z 798.972,A -85,B 0,C 180,E1 8463.501,E2 8463.501} C_VEL
LIN {X 0,Y 277.642,Z 818.057,A -85,B 0,C 180,E1 8462.234,E2 8462.234} C_VEL
LIN {X 0,Y 267.95,Z 836.564,A -85,B 0,C 180,E1 8460.653,E2 8460.653} C_VEL
LIN {X 0,Y 257.493,Z 853.823,A -85,B 0,C 180,E1 8458.769,E2 8458.769} C_VEL
LIN {X 0,Y 245.914,Z 870.5,A -85,B 0,C 180,E1 8456.427,E2 8456.427} C_VEL
LIN {X 0,Y 234.333,Z 885.353,A -85,B 0,C 180,E1 8453.745,E2 8453.745} C_VEL
LIN {X 0,Y 222.033,Z 899.453,A -85,B 0,C 180,E1 8450.427,E2 8450.427} C_VEL
LIN {X 0,Y 209.862,Z 912.02,A -85,B 0,C 180,E1 8446.499,E2 8446.499} C_VEL
LIN {X 0,Y 198.207,Z 923.01,A -85,B 0,C 180,E1 8441.883,E2 8441.883} C_VEL
LIN {X 0,Y 188.055,Z 931.919,A -85,B 0,C 180,E1 8436.83,E2 8436.83} C_VEL
LIN {X 0,Y 178.732,Z 939.702,A -85,B 0,C 180,E1 8430.756,E2 8430.756} C_VEL
LIN {X 0,Y 171.402,Z 945.614,A -85,B 0,C 180,E1 8424.164,E2 8424.164} C_VEL
LIN {X 0,Y 165.946,Z 949.939,A -85,B 0,C 180,E1 8416.794,E2 8416.794} C_VEL
LIN {X 0,Y 162.763,Z 952.379,A -85,B 0,C 180,E1 8409.282,E2 8409.282} C_VEL
LIN {X 0,Y 161.39,Z 953.197,A -85,B 0,C 180,E1 8401.921,E2 8401.921} C_VEL
LIN {X 0,Y 161.131,Z 952.736,A -85,B 0,C 180,E1 8395.342,E2 8395.342} C_VEL
LIN {X 0,Y 161.613,Z 950.954,A -85,B 0,C 180,E1 8388.758,E2 8388.758} C_VEL
LIN {X 0,Y 163.317,Z 947.616,A -85,B 0,C 180,E1 8381.603,E2 8381.603} C_VEL
LIN {X 0,Y 166.564,Z 942.859,A -85,B 0,C 180,E1 8374.803,E2 8374.803} C_VEL
LIN {X 0,Y 171.772,Z 936.059,A -85,B 0,C 180,E1 8367.991,E2 8367.991} C_VEL
LIN {X 0,Y 178.419,Z 927.829,A -85,B 0,C 180,E1 8361.94,E2 8361.94} C_VEL
LIN {X 0,Y 186.599,Z 917.749,A -85,B 0,C 180,E1 8356.357,E2 8356.357} C_VEL
LIN {X 0,Y 195.637,Z 906.261,A -85,B 0,C 180,E1 8351.52,E2 8351.52} C_VEL
LIN {X 0,Y 205.177,Z 893.413,A -85,B 0,C 180,E1 8347.352,E2 8347.352} C_VEL
LIN {X 0,Y 215.578,Z 878.18,A -85,B 0,C 180,E1 8343.555,E2 8343.555} C_VEL
LIN {X 0,Y 225.702,Z 861.695,A -85,B 0,C 180,E1 8340.395,E2 8340.395} C_VEL
LIN {X 0,Y 234.954,Z 844.732,A -85,B 0,C 180,E1 8337.858,E2 8337.858} C_VEL
LIN {X 0,Y 243.489,Z 826.94,A -85,B 0,C 180,E1 8335.761,E2 8335.761} C_VEL
LIN {X 0,Y 251.519,Z 807.48,A -85,B 0,C 180,E1 8333.956,E2 8333.956} C_VEL
LIN {X 0,Y 258.216,Z 788.178,A -85,B 0,C 180,E1 8332.555,E2 8332.555} C_VEL
LIN {X 0,Y 264.056,Z 767.362,A -85,B 0,C 180,E1 8331.399,E2 8331.399} C_VEL
LIN {X 0,Y 268.72,Z 745.401,A -85,B 0,C 180,E1 8330.508,E2 8330.508} C_VEL
LIN {X 0,Y 271.875,Z 723.796,A -85,B 0,C 180,E1 8329.902,E2 8329.902} C_VEL
LIN {X 0,Y 285.103,Z 593.487,A -85,B 0,C 180,E1 8327.124,E2 8327.124} C_VEL
LIN {X 0,Y 280.107,Z 583.874,A -85,B 0,C 180,E1 8323.971,E2 8323.971} C_VEL
LIN {X 0,Y 274.544,Z 573.74,A -85,B 0,C 180,E1 8319.865,E2 8319.865} C_VEL
LIN {X 0,Y 270.749,Z 567.497,A -85,B 0,C 180,E1 8316.548,E2 8316.548} C_VEL
LIN {X 0,Y 268.582,Z 563.968,A -85,B 0,C 180,E1 8314.333,E2 8314.333} C_VEL
LIN {X 0,Y 266.586,Z 560.565,A -85,B 0,C 180,E1 8311.928,E2 8311.928} C_VEL
LIN {X 0,Y 264.095,Z 556.496,A -85,B 0,C 180,E1 8308.246,E2 8308.246} C_VEL
LIN {X 0,Y 261.563,Z 552.37,A -85,B 0,C 180,E1 8302.238,E2 8302.238} C_VEL
LIN {X 0,Y 260.805,Z 551.633,A -85,B 0,C 180,E1 8296.94,E2 8296.94} C_VEL
LIN {X 0,Y 261.548,Z 552.318,A -85,B 0,C 180,E1 8291.69,E2 8291.69} C_VEL
LIN {X 0,Y 262.244,Z 553.637,A -85,B 0,C 180,E1 8289.437,E2 8289.437} C_VEL
LIN {X 0,Y 264.966,Z 557.614,A -85,B 0,C 180,E1 8284.22,E2 8284.22} C_VEL
LIN {X 0,Y 268.113,Z 562.608,A -85,B 0,C 180,E1 8280.107,E2 8280.107} C_VEL
LIN {X 0,Y 271.286,Z 567.733,A -85,B 0,C 180,E1 8276.831,E2 8276.831} C_VEL
LIN {X 0,Y 275.397,Z 574.311,A -85,B 0,C 180,E1 8273.329,E2 8273.329} C_VEL
LIN {X 0,Y 280.784,Z 583.763,A -85,B 0,C 180,E1 8269.433,E2 8269.433} C_VEL
LIN {X 0,Y 286.182,Z 593.568,A -85,B 0,C 180,E1 8266.102,E2 8266.102} C_VEL
LIN {X 0,Y 288.315,Z 597.695,A -85,B 0,C 180,E1 8264.887,E2 8264.887} C_VEL
LIN {X 0,Y 288.641,Z 599.763,A -85,B 0,C 180,E1 8264.619,E2 8264.619} C_VEL
LIN {X 0,Y 288.272,Z 603.109,A -85,B 0,C 180,E1 8264.571,E2 8264.571} C_VEL
LIN {X 0,Y 286.979,Z 607.952,A -85,B 0,C 180,E1 8264.826,E2 8264.826} C_VEL
LIN {X 0,Y 284.138,Z 616.66,A -85,B 0,C 180,E1 8265.53,E2 8265.53} C_VEL
LIN {X 0,Y 283.366,Z 620.906,A -85,B 0,C 180,E1 8265.602,E2 8265.602} C_VEL
LIN {X 0,Y 270.985,Z 745.939,A -85,B 0,C 180,E1 8262.992,E2 8262.992} C_VEL
LIN {X 0,Y 267.054,Z 768.196,A -85,B 0,C 180,E1 8262.348,E2 8262.348} C_VEL
LIN {X 0,Y 261.691,Z 789.557,A -85,B 0,C 180,E1 8261.542,E2 8261.542} C_VEL
LIN {X 0,Y 254.726,Z 811.378,A -85,B 0,C 180,E1 8260.409,E2 8260.409} C_VEL
LIN {X 0,Y 247.285,Z 830.698,A -85,B 0,C 180,E1 8259.078,E2 8259.078} C_VEL
LIN {X 0,Y 238.395,Z 850.234,A -85,B 0,C 180,E1 8257.334,E2 8257.334} C_VEL
LIN {X 0,Y 228.996,Z 868.131,A -85,B 0,C 180,E1 8255.264,E2 8255.264} C_VEL
LIN {X 0,Y 218.451,Z 885.911,A -85,B 0,C 180,E1 8252.625,E2 8252.625} C_VEL
LIN {X 0,Y 208.185,Z 901.583,A -85,B 0,C 180,E1 8249.626,E2 8249.626} C_VEL
LIN {X 0,Y 197.728,Z 916.156,A -85,B 0,C 180,E1 8246.036,E2 8246.036} C_VEL
LIN {X 0,Y 187.308,Z 929.676,A -85,B 0,C 180,E1 8241.7,E2 8241.7} C_VEL
LIN {X 0,Y 177.043,Z 942.453,A -85,B 0,C 180,E1 8236.301,E2 8236.301} C_VEL
LIN {X 0,Y 168.416,Z 953.09,A -85,B 0,C 180,E1 8230.332,E2 8230.332} C_VEL
LIN {X 0,Y 161.313,Z 962.247,A -85,B 0,C 180,E1 8223.488,E2 8223.488} C_VEL
LIN {X 0,Y 156.375,Z 969.398,A -85,B 0,C 180,E1 8216.187,E2 8216.187} C_VEL
LIN {X 0,Y 153.497,Z 975.047,A -85,B 0,C 180,E1 8208.228,E2 8208.228} C_VEL
LIN {X 0,Y 152.663,Z 978.683,A -85,B 0,C 180,E1 8200.766,E2 8200.766} C_VEL
LIN {X 0,Y 152.855,Z 980.408,A -85,B 0,C 180,E1 8194.51,E2 8194.51} C_VEL
LIN {X 0,Y 152.996,Z 980.977,A -85,B 0,C 180,E1 8189.634,E2 8189.634} C_VEL
LIN {X 0,Y 152.762,Z 980.761,A -85,B 0,C 180,E1 8184.374,E2 8184.374} C_VEL
LIN {X 0,Y 152.645,Z 979.332,A -85,B 0,C 180,E1 8177.413,E2 8177.413} C_VEL
LIN {X 0,Y 154.014,Z 976.08,A -85,B 0,C 180,E1 8169.487,E2 8169.487} C_VEL
LIN {X 0,Y 157.847,Z 970.957,A -85,B 0,C 180,E1 8161.232,E2 8161.232} C_VEL
LIN {X 0,Y 164.385,Z 964.019,A -85,B 0,C 180,E1 8153.404,E2 8153.404} C_VEL
LIN {X 0,Y 173.508,Z 955.097,A -85,B 0,C 180,E1 8146.261,E2 8146.261} C_VEL
LIN {X 0,Y 184.324,Z 944.731,A -85,B 0,C 180,E1 8140.203,E2 8140.203} C_VEL
LIN {X 0,Y 196.562,Z 932.748,A -85,B 0,C 180,E1 8135.032,E2 8135.032} C_VEL
LIN {X 0,Y 208.704,Z 920.236,A -85,B 0,C 180,E1 8130.971,E2 8130.971} C_VEL
LIN {X 0,Y 222.09,Z 905.315,A -85,B 0,C 180,E1 8127.335,E2 8127.335} C_VEL
LIN {X 0,Y 234.984,Z 889.505,A -85,B 0,C 180,E1 8124.432,E2 8124.432} C_VEL
LIN {X 0,Y 247.381,Z 872.666,A -85,B 0,C 180,E1 8122.078,E2 8122.078} C_VEL
LIN {X 0,Y 258.849,Z 855.223,A -85,B 0,C 180,E1 8120.194,E2 8120.194} C_VEL
LIN {X 0,Y 269.149,Z 837.251,A -85,B 0,C 180,E1 8118.704,E2 8118.704} C_VEL
LIN {X 0,Y 278.779,Z 817.779,A -85,B 0,C 180,E1 8117.461,E2 8117.461} C_VEL
LIN {X 0,Y 287.243,Z 797.492,A -85,B 0,C 180,E1 8116.489,E2 8116.489} C_VEL
LIN {X 0,Y 294.044,Z 777.608,A -85,B 0,C 180,E1 8115.785,E2 8115.785} C_VEL
LIN {X 0,Y 299.948,Z 754.848,A -85,B 0,C 180,E1 8115.174,E2 8115.174} C_VEL
LIN {X 0,Y 303.85,Z 733.09,A -85,B 0,C 180,E1 8114.706,E2 8114.706} C_VEL
LIN {X 0,Y 318.221,Z 621.891,A -85,B 0,C 180,E1 8112.571,E2 8112.571} C_VEL
LIN {X 0,Y 318.113,Z 621.135,A -85,B 0,C 180,E1 8111.42,E2 8111.42} C_VEL
LIN {X 0,Y 318.097,Z 621.32,A -85,B 0,C 180,E1 8110.138,E2 8110.138} C_VEL
LIN {X 0,Y 318.06,Z 622.009,A -85,B 0,C 180,E1 8109.61,E2 8109.61} C_VEL
LIN {X 0,Y 302.458,Z 738.205,A -85,B 0,C 180,E1 8107.418,E2 8107.418} C_VEL
LIN {X 0,Y 297.924,Z 759.3,A -85,B 0,C 180,E1 8106.841,E2 8106.841} C_VEL
LIN {X 0,Y 292.1,Z 779.384,A -85,B 0,C 180,E1 8106.091,E2 8106.091} C_VEL
LIN {X 0,Y 284.813,Z 799.266,A -85,B 0,C 180,E1 8105.114,E2 8105.114} C_VEL
LIN {X 0,Y 276.548,Z 817.779,A -85,B 0,C 180,E1 8103.938,E2 8103.938} C_VEL
LIN {X 0,Y 266.673,Z 836.285,A -85,B 0,C 180,E1 8102.435,E2 8102.435} C_VEL
LIN {X 0,Y 255.95,Z 853.568,A -85,B 0,C 180,E1 8100.632,E2 8100.632} C_VEL
LIN {X 0,Y 243.896,Z 870.516,A -85,B 0,C 180,E1 8098.355,E2 8098.355} C_VEL
LIN {X 0,Y 232.088,Z 885.2,A -85,B 0,C 180,E1 8095.799,E2 8095.799} C_VEL
LIN {X 0,Y 219.279,Z 899.363,A -85,B 0,C 180,E1 8092.577,E2 8092.577} C_VEL
LIN {X 0,Y 206.846,Z 911.658,A -85,B 0,C 180,E1 8088.851,E2 8088.851} C_VEL
LIN {X 0,Y 195.019,Z 922.376,A -85,B 0,C 180,E1 8084.522,E2 8084.522} C_VEL
LIN {X 0,Y 183.572,Z 931.934,A -85,B 0,C 180,E1 8079.265,E2 8079.265} C_VEL
LIN {X 0,Y 173.658,Z 939.709,A -85,B 0,C 180,E1 8073.313,E2 8073.313} C_VEL
LIN {X 0,Y 164.965,Z 946.168,A -85,B 0,C 180,E1 8066.108,E2 8066.108} C_VEL
LIN {X 0,Y 158.857,Z 950.511,A -85,B 0,C 180,E1 8058.49,E2 8058.49} C_VEL
LIN {X 0,Y 155.31,Z 952.945,A -85,B 0,C 180,E1 8051.033,E2 8051.033} C_VEL
LIN {X 0,Y 153.554,Z 953.934,A -85,B 0,C 180,E1 8043.148,E2 8043.148} C_VEL
LIN {X 0,Y 153.154,Z 953.58,A -85,B 0,C 180,E1 8036.566,E2 8036.566} C_VEL
LIN {X 0,Y 153.544,Z 951.933,A -85,B 0,C 180,E1 8029.388,E2 8029.388} C_VEL
LIN {X 0,Y 155.081,Z 949.023,A -85,B 0,C 180,E1 8022.276,E2 8022.276} C_VEL
LIN {X 0,Y 158.507,Z 944.11,A -85,B 0,C 180,E1 8014.672,E2 8014.672} C_VEL
LIN {X 0,Y 163.542,Z 937.861,A -85,B 0,C 180,E1 8007.89,E2 8007.89} C_VEL
LIN {X 0,Y 170.725,Z 929.473,A -85,B 0,C 180,E1 8001.235,E2 8001.235} C_VEL
LIN {X 0,Y 179.187,Z 919.618,A -85,B 0,C 180,E1 7995.451,E2 7995.451} C_VEL
LIN {X 0,Y 188.526,Z 908.376,A -85,B 0,C 180,E1 7990.474,E2 7990.474} C_VEL
LIN {X 0,Y 198.963,Z 894.924,A -85,B 0,C 180,E1 7985.974,E2 7985.974} C_VEL
LIN {X 0,Y 209.053,Z 880.728,A -85,B 0,C 180,E1 7982.353,E2 7982.353} C_VEL
LIN {X 0,Y 219.102,Z 865.15,A -85,B 0,C 180,E1 7979.257,E2 7979.257} C_VEL
LIN {X 0,Y 228.934,Z 848.066,A -85,B 0,C 180,E1 7976.607,E2 7976.607} C_VEL
LIN {X 0,Y 238.052,Z 830.03,A -85,B 0,C 180,E1 7974.423,E2 7974.423} C_VEL
LIN {X 0,Y 246.282,Z 811.144,A -85,B 0,C 180,E1 7972.626,E2 7972.626} C_VEL
LIN {X 0,Y 253.51,Z 791.264,A -85,B 0,C 180,E1 7971.158,E2 7971.158} C_VEL
LIN {X 0,Y 259.477,Z 771.023,A -85,B 0,C 180,E1 7970.013,E2 7970.013} C_VEL
LIN {X 0,Y 264.417,Z 749.414,A -85,B 0,C 180,E1 7969.102,E2 7969.102} C_VEL
LIN {X 0,Y 268.053,Z 726.718,A -85,B 0,C 180,E1 7968.438,E2 7968.438} C_VEL
LIN {X 0,Y 281.483,Z 597.957,A -85,B 0,C 180,E1 7965.706,E2 7965.706} C_VEL
LIN {X 0,Y 276.153,Z 587.523,A -85,B 0,C 180,E1 7962.054,E2 7962.054} C_VEL
LIN {X 0,Y 271.874,Z 579.721,A -85,B 0,C 180,E1 7958.63,E2 7958.63} C_VEL
LIN {X 0,Y 267.884,Z 572.804,A -85,B 0,C 180,E1 7954.796,E2 7954.796} C_VEL
LIN {X 0,Y 265.153,Z 568.234,A -85,B 0,C 180,E1 7951.54,E2 7951.54} C_VEL
LIN {X 0,Y 262.788,Z 564.25,A -85,B 0,C 180,E1 7947.905,E2 7947.905} C_VEL
LIN {X 0,Y 260.451,Z 560.271,A -85,B 0,C 180,E1 7942.1,E2 7942.1} C_VEL
LIN {X 0,Y 259.732,Z 559.555,A -85,B 0,C 180,E1 7936.782,E2 7936.782} C_VEL
LIN {X 0,Y 260.603,Z 560.352,A -85,B 0,C 180,E1 7931.285,E2 7931.285} C_VEL
LIN {X 0,Y 263.637,Z 565.345,A -85,B 0,C 180,E1 7924.569,E2 7924.569} C_VEL
LIN {X 0,Y 266.61,Z 570.21,A -85,B 0,C 180,E1 7920.538,E2 7920.538} C_VEL
LIN {X 0,Y 269.699,Z 575.359,A -85,B 0,C 180,E1 7917.238,E2 7917.238} C_VEL
LIN {X 0,Y 273.55,Z 581.708,A -85,B 0,C 180,E1 7913.847,E2 7913.847} C_VEL
LIN {X 0,Y 278.889,Z 591.307,A -85,B 0,C 180,E1 7909.883,E2 7909.883} C_VEL
LIN {X 0,Y 284.106,Z 601.086,A -85,B 0,C 180,E1 7906.57,E2 7906.57} C_VEL
LIN {X 0,Y 285.114,Z 603.33,A -85,B 0,C 180,E1 7905.954,E2 7905.954} C_VEL
LIN {X 0,Y 283.366,Z 620.906,A -85,B 0,C 180,E1 7905.602,E2 7905.602} C_VEL
LIN {X 0,Y 282.201,Z 628.582,A -85,B 0,C 180,E1 7905.631,E2 7905.631} C_VEL
LIN {X 0,Y 277.622,Z 648.999,A -85,B 0,C 180,E1 7906.388,E2 7906.388} C_VEL
LIN {X 0,Y 276.65,Z 655.588,A -85,B 0,C 180,E1 7906.397,E2 7906.397} C_VEL
LIN {X 0,Y 267.483,Z 745.648,A -85,B 0,C 180,E1 7904.527,E2 7904.527} C_VEL
LIN {X 0,Y 263.457,Z 767.934,A -85,B 0,C 180,E1 7903.895,E2 7903.895} C_VEL
LIN {X 0,Y 258.093,Z 788.892,A -85,B 0,C 180,E1 7903.124,E2 7903.124} C_VEL
LIN {X 0,Y 251.199,Z 810.167,A -85,B 0,C 180,E1 7902.056,E2 7902.056} C_VEL
LIN {X 0,Y 243.588,Z 829.623,A -85,B 0,C 180,E1 7900.759,E2 7900.759} C_VEL
LIN {X 0,Y 234.476,Z 849.203,A -85,B 0,C 180,E1 7899.055,E2 7899.055} C_VEL
LIN {X 0,Y 224.82,Z 867.182,A -85,B 0,C 180,E1 7897.025,E2 7897.025} C_VEL
LIN {X 0,Y 213.956,Z 885.057,A -85,B 0,C 180,E1 7894.422,E2 7894.422} C_VEL
LIN {X 0,Y 203.167,Z 901.036,A -85,B 0,C 180,E1 7891.397,E2 7891.397} C_VEL
LIN {X 0,Y 191.813,Z 916.309,A -85,B 0,C 180,E1 7887.623,E2 7887.623} C_VEL
LIN {X 0,Y 180.996,Z 929.695,A -85,B 0,C 180,E1 7883.236,E2 7883.236} C_VEL
LIN {X 0,Y 170.813,Z 941.744,A -85,B 0,C 180,E1 7878.03,E2 7878.03} C_VEL
LIN {X 0,Y 161.675,Z 952.403,A -85,B 0,C 180,E1 7871.915,E2 7871.915} C_VEL
LIN {X 0,Y 154.088,Z 961.577,A -85,B 0,C 180,E1 7864.83,E2 7864.83} C_VEL
LIN {X 0,Y 148.76,Z 968.728,A -85,B 0,C 180,E1 7857.205,E2 7857.205} C_VEL
LIN {X 0,Y 145.621,Z 974.368,A -85,B 0,C 180,E1 7848.835,E2 7848.835} C_VEL
LIN {X 0,Y 144.694,Z 977.94,A -85,B 0,C 180,E1 7841.12,E2 7841.12} C_VEL
LIN {X 0,Y 144.892,Z 979.703,A -85,B 0,C 180,E1 7834.362,E2 7834.362} C_VEL
LIN {X 0,Y 145.019,Z 980.251,A -85,B 0,C 180,E1 7829.218,E2 7829.218} C_VEL
LIN {X 0,Y 144.731,Z 980.001,A -85,B 0,C 180,E1 7823.663,E2 7823.663} C_VEL
LIN {X 0,Y 144.72,Z 978.57,A -85,B 0,C 180,E1 7816.423,E2 7816.423} C_VEL
LIN {X 0,Y 146.446,Z 975.26,A -85,B 0,C 180,E1 7807.954,E2 7807.954} C_VEL
LIN {X 0,Y 151.143,Z 969.832,A -85,B 0,C 180,E1 7798.947,E2 7798.947} C_VEL
LIN {X 0,Y 158.147,Z 963.184,A -85,B 0,C 180,E1 7791.262,E2 7791.262} C_VEL
LIN {X 0,Y 168.091,Z 954.269,A -85,B 0,C 180,E1 7783.979,E2 7783.979} C_VEL
LIN {X 0,Y 179.776,Z 943.825,A -85,B 0,C 180,E1 7777.85,E2 7777.85} C_VEL
LIN {X 0,Y 193.199,Z 931.382,A -85,B 0,C 180,E1 7772.562,E2 7772.562} C_VEL
LIN {X 0,Y 206.06,Z 918.732,A -85,B 0,C 180,E1 7768.582,E2 7768.582} C_VEL
LIN {X 0,Y 219.757,Z 904.076,A -85,B 0,C 180,E1 7765.138,E2 7765.138} C_VEL
LIN {X 0,Y 232.573,Z 888.874,A -85,B 0,C 180,E1 7762.454,E2 7762.454} C_VEL
LIN {X 0,Y 245.917,Z 871.322,A -85,B 0,C 180,E1 7760.1,E2 7760.1} C_VEL
LIN {X 0,Y 257.607,Z 853.915,A -85,B 0,C 180,E1 7758.323,E2 7758.323} C_VEL
LIN {X 0,Y 268.323,Z 835.68,A -85,B 0,C 180,E1 7756.896,E2 7756.896} C_VEL
LIN {X 0,Y 277.428,Z 817.604,A -85,B 0,C 180,E1 7755.811,E2 7755.811} C_VEL
LIN {X 0,Y 286.043,Z 797.536,A -85,B 0,C 180,E1 7754.896,E2 7754.896} C_VEL
LIN {X 0,Y 293.387,Z 776.524,A -85,B 0,C 180,E1 7754.195,E2 7754.195} C_VEL
LIN {X 0,Y 299.263,Z 754.225,A -85,B 0,C 180,E1 7753.63,E2 7753.63} C_VEL
LIN {X 0,Y 303.288,Z 732.128,A -85,B 0,C 180,E1 7753.177,E2 7753.177} C_VEL
LIN {X 0,Y 317.018,Z 629.05,A -85,B 0,C 180,E1 7751.251,E2 7751.251} C_VEL
LIN {X 0,Y 316.987,Z 629.233,A -85,B 0,C 180,E1 7750.932,E2 7750.932} C_VEL
LIN {X 0,Y 301.918,Z 738.636,A -85,B 0,C 180,E1 7748.931,E2 7748.931} C_VEL
LIN {X 0,Y 297.322,Z 759.706,A -85,B 0,C 180,E1 7748.381,E2 7748.381} C_VEL
LIN {X 0,Y 291.301,Z 780.024,A -85,B 0,C 180,E1 7747.657,E2 7747.657} C_VEL
LIN {X 0,Y 283.886,Z 799.745,A -85,B 0,C 180,E1 7746.729,E2 7746.729} C_VEL
LIN {X 0,Y 275.235,Z 818.653,A -85,B 0,C 180,E1 7745.58,E2 7745.58} C_VEL
LIN {X 0,Y 265.125,Z 837.064,A -85,B 0,C 180,E1 7744.142,E2 7744.142} C_VEL
LIN {X 0,Y 254.161,Z 854.202,A -85,B 0,C 180,E1 7742.42,E2 7742.42} C_VEL
LIN {X 0,Y 242.441,Z 870.269,A -85,B 0,C 180,E1 7740.356,E2 7740.356} C_VEL
LIN {X 0,Y 230.097,Z 885.188,A -85,B 0,C 180,E1 7737.873,E2 7737.873} C_VEL
LIN {X 0,Y 217.351,Z 898.789,A -85,B 0,C 180,E1 7734.902,E2 7734.902} C_VEL
LIN {X 0,Y 204.247,Z 911.349,A -85,B 0,C 180,E1 7731.27,E2 7731.27} C_VEL
LIN {X 0,Y 191.021,Z 922.798,A -85,B 0,C 180,E1 7726.764,E2 7726.764} C_VEL
LIN {X 0,Y 179.073,Z 932.262,A -85,B 0,C 180,E1 7721.632,E2 7721.632} C_VEL
LIN {X 0,Y 167.943,Z 940.405,A -85,B 0,C 180,E1 7715.369,E2 7715.369} C_VEL
LIN {X 0,Y 158.747,Z 946.691,A -85,B 0,C 180,E1 7708.225,E2 7708.225} C_VEL
LIN {X 0,Y 151.901,Z 951.113,A -85,B 0,C 180,E1 7700.32,E2 7700.32} C_VEL
LIN {X 0,Y 147.807,Z 953.623,A -85,B 0,C 180,E1 7692.493,E2 7692.493} C_VEL
LIN {X 0,Y 145.774,Z 954.677,A -85,B 0,C 180,E1 7684.604,E2 7684.604} C_VEL
LIN {X 0,Y 145.205,Z 954.415,A -85,B 0,C 180,E1 7677.91,E2 7677.91} C_VEL
LIN {X 0,Y 145.455,Z 953.042,A -85,B 0,C 180,E1 7670.513,E2 7670.513} C_VEL
LIN {X 0,Y 146.856,Z 950.269,A -85,B 0,C 180,E1 7662.975,E2 7662.975} C_VEL
LIN {X 0,Y 149.983,Z 945.897,A -85,B 0,C 180,E1 7655.347,E2 7655.347} C_VEL
LIN {X 0,Y 155.303,Z 939.646,A -85,B 0,C 180,E1 7647.778,E2 7647.778} C_VEL
LIN {X 0,Y 162.233,Z 932.033,A -85,B 0,C 180,E1 7641.129,E2 7641.129} C_VEL
LIN {X 0,Y 170.823,Z 922.543,A -85,B 0,C 180,E1 7635.069,E2 7635.069} C_VEL
LIN {X 0,Y 180.332,Z 911.659,A -85,B 0,C 180,E1 7629.887,E2 7629.887} C_VEL
LIN {X 0,Y 190.363,Z 899.487,A -85,B 0,C 180,E1 7625.478,E2 7625.478} C_VEL
LIN {X 0,Y 200.621,Z 886.057,A -85,B 0,C 180,E1 7621.735,E2 7621.735} C_VEL
LIN {X 0,Y 211.154,Z 870.886,A -85,B 0,C 180,E1 7618.468,E2 7618.468} C_VEL
LIN {X 0,Y 221.569,Z 853.939,A -85,B 0,C 180,E1 7615.656,E2 7615.656} C_VEL
LIN {X 0,Y 230.702,Z 837.074,A -85,B 0,C 180,E1 7613.477,E2 7613.477} C_VEL
LIN {X 0,Y 239.61,Z 818.122,A -85,B 0,C 180,E1 7611.551,E2 7611.551} C_VEL
LIN {X 0,Y 247.383,Z 798.596,A -85,B 0,C 180,E1 7610.006,E2 7610.006} C_VEL
LIN {X 0,Y 254.038,Z 778.297,A -85,B 0,C 180,E1 7608.767,E2 7608.767} C_VEL
LIN {X 0,Y 259.612,Z 756.576,A -85,B 0,C 180,E1 7607.778,E2 7607.778} C_VEL
LIN {X 0,Y 263.657,Z 734.689,A -85,B 0,C 180,E1 7607.068,E2 7607.068} C_VEL
LIN {X 0,Y 267.91,Z 697.823,A -85,B 0,C 180,E1 7606.257,E2 7606.257} C_VEL
LIN {X 0,Y 278.031,Z 602.494,A -85,B 0,C 180,E1 7604.299,E2 7604.299} C_VEL
LIN {X 0,Y 272.404,Z 591.432,A -85,B 0,C 180,E1 7600.104,E2 7600.104} C_VEL
LIN {X 0,Y 268.455,Z 584.188,A -85,B 0,C 180,E1 7596.579,E2 7596.579} C_VEL
LIN {X 0,Y 265.641,Z 579.33,A -85,B 0,C 180,E1 7593.594,E2 7593.594} C_VEL
LIN {X 0,Y 263.656,Z 575.799,A -85,B 0,C 180,E1 7591.048,E2 7591.048} C_VEL
LIN {X 0,Y 261.432,Z 571.933,A -85,B 0,C 180,E1 7587.458,E2 7587.458} C_VEL
LIN {X 0,Y 259.339,Z 568.171,A -85,B 0,C 180,E1 7581.962,E2 7581.962} C_VEL
LIN {X 0,Y 258.663,Z 567.474,A -85,B 0,C 180,E1 7576.526,E2 7576.526} C_VEL
LIN {X 0,Y 259.513,Z 568.282,A -85,B 0,C 180,E1 7571.333,E2 7571.333} C_VEL
LIN {X 0,Y 262.315,Z 573.075,A -85,B 0,C 180,E1 7564.921,E2 7564.921} C_VEL
LIN {X 0,Y 265.205,Z 577.977,A -85,B 0,C 180,E1 7560.865,E2 7560.865} C_VEL
LIN {X 0,Y 268.121,Z 582.982,A -85,B 0,C 180,E1 7557.65,E2 7557.65} C_VEL
LIN {X 0,Y 271.802,Z 589.262,A -85,B 0,C 180,E1 7554.3,E2 7554.3} C_VEL
LIN {X 0,Y 277.201,Z 599.22,A -85,B 0,C 180,E1 7550.188,E2 7550.188} C_VEL
LIN {X 0,Y 281.5,Z 607.603,A -85,B 0,C 180,E1 7547.355,E2 7547.355} C_VEL
LIN {X 0,Y 276.65,Z 655.588,A -85,B 0,C 180,E1 7546.397,E2 7546.397} C_VEL
LIN {X 0,Y 275.466,Z 663.265,A -85,B 0,C 180,E1 7546.434,E2 7546.434} C_VEL
LIN {X 0,Y 270.901,Z 683.675,A -85,B 0,C 180,E1 7547.228,E2 7547.228} C_VEL
LIN {X 0,Y 269.949,Z 690.264,A -85,B 0,C 180,E1 7547.236,E2 7547.236} C_VEL
LIN {X 0,Y 263.983,Z 746.024,A -85,B 0,C 180,E1 7546.076,E2 7546.076} C_VEL
LIN {X 0,Y 259.859,Z 768.249,A -85,B 0,C 180,E1 7545.458,E2 7545.458} C_VEL
LIN {X 0,Y 254.273,Z 789.439,A -85,B 0,C 180,E1 7544.694,E2 7544.694} C_VEL
LIN {X 0,Y 247.446,Z 809.98,A -85,B 0,C 180,E1 7543.683,E2 7543.683} C_VEL
LIN {X 0,Y 239.675,Z 829.402,A -85,B 0,C 180,E1 7542.42,E2 7542.42} C_VEL
LIN {X 0,Y 230.211,Z 849.281,A -85,B 0,C 180,E1 7540.727,E2 7540.727} C_VEL
LIN {X 0,Y 220.141,Z 867.477,A -85,B 0,C 180,E1 7538.695,E2 7538.695} C_VEL
LIN {X 0,Y 209.289,Z 884.752,A -85,B 0,C 180,E1 7536.198,E2 7536.198} C_VEL
LIN {X 0,Y 198.246,Z 900.566,A -85,B 0,C 180,E1 7533.225,E2 7533.225} C_VEL
LIN {X 0,Y 186.745,Z 915.49,A -85,B 0,C 180,E1 7529.553,E2 7529.553} C_VEL
LIN {X 0,Y 175.453,Z 928.937,A -85,B 0,C 180,E1 7525.156,E2 7525.156} C_VEL
LIN {X 0,Y 164.75,Z 941.028,A -85,B 0,C 180,E1 7519.888,E2 7519.888} C_VEL
LIN {X 0,Y 155.435,Z 951.31,A -85,B 0,C 180,E1 7513.909,E2 7513.909} C_VEL
LIN {X 0,Y 147.304,Z 960.445,A -85,B 0,C 180,E1 7506.687,E2 7506.687} C_VEL
LIN {X 0,Y 141.426,Z 967.711,A -85,B 0,C 180,E1 7498.743,E2 7498.743} C_VEL
LIN {X 0,Y 137.867,Z 973.456,A -85,B 0,C 180,E1 7489.938,E2 7489.938} C_VEL
LIN {X 0,Y 136.727,Z 977.194,A -85,B 0,C 180,E1 7481.509,E2 7481.509} C_VEL
LIN {X 0,Y 136.912,Z 978.927,A -85,B 0,C 180,E1 7474.616,E2 7474.616} C_VEL
LIN {X 0,Y 137.052,Z 979.512,A -85,B 0,C 180,E1 7469.173,E2 7469.173} C_VEL
LIN {X 0,Y 136.758,Z 979.335,A -85,B 0,C 180,E1 7463.713,E2 7463.713} C_VEL
LIN {X 0,Y 136.73,Z 978.078,A -85,B 0,C 180,E1 7456.477,E2 7456.477} C_VEL
LIN {X 0,Y 138.665,Z 974.829,A -85,B 0,C 180,E1 7447.095,E2 7447.095} C_VEL
LIN {X 0,Y 143.248,Z 970.105,A -85,B 0,C 180,E1 7438.378,E2 7438.378} C_VEL
LIN {X 0,Y 150.89,Z 963.395,A -85,B 0,C 180,E1 7430.014,E2 7430.014} C_VEL
LIN {X 0,Y 161.353,Z 954.744,A -85,B 0,C 180,E1 7422.487,E2 7422.487} C_VEL
LIN {X 0,Y 174.169,Z 944.109,A -85,B 0,C 180,E1 7415.973,E2 7415.973} C_VEL
LIN {X 0,Y 187.554,Z 932.53,A -85,B 0,C 180,E1 7410.89,E2 7410.89} C_VEL
LIN {X 0,Y 202.266,Z 918.836,A -85,B 0,C 180,E1 7406.543,E2 7406.543} C_VEL
LIN {X 0,Y 216.422,Z 904.291,A -85,B 0,C 180,E1 7403.185,E2 7403.185} C_VEL
LIN {X 0,Y 230.034,Z 888.867,A -85,B 0,C 180,E1 7400.518,E2 7400.518} C_VEL
LIN {X 0,Y 243.715,Z 871.492,A -85,B 0,C 180,E1 7398.263,E2 7398.263} C_VEL
LIN {X 0,Y 255.573,Z 854.51,A -85,B 0,C 180,E1 7396.588,E2 7396.588} C_VEL
LIN {X 0,Y 267.219,Z 835.193,A -85,B 0,C 180,E1 7395.148,E2 7395.148} C_VEL
LIN {X 0,Y 276.776,Z 816.683,A -85,B 0,C 180,E1 7394.105,E2 7394.105} C_VEL
LIN {X 0,Y 285.535,Z 796.553,A -85,B 0,C 180,E1 7393.253,E2 7393.253} C_VEL
LIN {X 0,Y 292.694,Z 776.515,A -85,B 0,C 180,E1 7392.628,E2 7392.628} C_VEL
LIN {X 0,Y 298.657,Z 754.552,A -85,B 0,C 180,E1 7392.1,E2 7392.1} C_VEL
LIN {X 0,Y 302.842,Z 732.584,A -85,B 0,C 180,E1 7391.669,E2 7391.669} C_VEL
LIN {X 0,Y 307.023,Z 702.192,A -85,B 0,C 180,E1 7391.12,E2 7391.12} C_VEL
LIN {X 0,Y 301.392,Z 740.727,A -85,B 0,C 180,E1 7390.414,E2 7390.414} C_VEL
LIN {X 0,Y 296.612,Z 761.772,A -85,B 0,C 180,E1 7389.878,E2 7389.878} C_VEL
LIN {X 0,Y 290.402,Z 781.803,A -85,B 0,C 180,E1 7389.185,E2 7389.185} C_VEL
LIN {X 0,Y 282.35,Z 802.327,A -85,B 0,C 180,E1 7388.247,E2 7388.247} C_VEL
LIN {X 0,Y 273.455,Z 820.992,A -85,B 0,C 180,E1 7387.141,E2 7387.141} C_VEL
LIN {X 0,Y 262.916,Z 839.474,A -85,B 0,C 180,E1 7385.733,E2 7385.733} C_VEL
LIN {X 0,Y 251.565,Z 856.501,A -85,B 0,C 180,E1 7384.057,E2 7384.057} C_VEL
LIN {X 0,Y 239.081,Z 872.783,A -85,B 0,C 180,E1 7381.986,E2 7381.986} C_VEL
LIN {X 0,Y 225.949,Z 887.884,A -85,B 0,C 180,E1 7379.474,E2 7379.474} C_VEL
LIN {X 0,Y 212.354,Z 901.708,A -85,B 0,C 180,E1 7376.43,E2 7376.43} C_VEL
LIN {X 0,Y 198.541,Z 914.153,A -85,B 0,C 180,E1 7372.728,E2 7372.728} C_VEL
LIN {X 0,Y 185.269,Z 924.891,A -85,B 0,C 180,E1 7368.343,E2 7368.343} C_VEL
LIN {X 0,Y 172.489,Z 934.271,A -85,B 0,C 180,E1 7362.997,E2 7362.997} C_VEL
LIN {X 0,Y 161.088,Z 941.98,A -85,B 0,C 180,E1 7356.702,E2 7356.702} C_VEL
LIN {X 0,Y 151.611,Z 947.939,A -85,B 0,C 180,E1 7349.481,E2 7349.481} C_VEL
LIN {X 0,Y 144.473,Z 952.125,A -85,B 0,C 180,E1 7341.432,E2 7341.432} C_VEL
LIN {X 0,Y 140.058,Z 954.489,A -85,B 0,C 180,E1 7333.248,E2 7333.248} C_VEL
LIN {X 0,Y 137.775,Z 955.422,A -85,B 0,C 180,E1 7324.464,E2 7324.464} C_VEL
LIN {X 0,Y 137.221,Z 955.046,A -85,B 0,C 180,E1 7317.255,E2 7317.255} C_VEL
LIN {X 0,Y 137.575,Z 953.48,A -85,B 0,C 180,E1 7309.521,E2 7309.521} C_VEL
LIN {X 0,Y 139.252,Z 950.611,A -85,B 0,C 180,E1 7301.589,E2 7301.589} C_VEL
LIN {X 0,Y 143.073,Z 945.768,A -85,B 0,C 180,E1 7293.196,E2 7293.196} C_VEL
LIN {X 0,Y 148.737,Z 939.581,A -85,B 0,C 180,E1 7285.751,E2 7285.751} C_VEL
LIN {X 0,Y 156.292,Z 931.752,A -85,B 0,C 180,E1 7278.927,E2 7278.927} C_VEL
LIN {X 0,Y 165.543,Z 922.103,A -85,B 0,C 180,E1 7272.778,E2 7272.778} C_VEL
LIN {X 0,Y 176.263,Z 910.351,A -85,B 0,C 180,E1 7267.304,E2 7267.304} C_VEL
LIN {X 0,Y 186.892,Z 897.758,A -85,B 0,C 180,E1 7262.945,E2 7262.945} C_VEL
LIN {X 0,Y 197.844,Z 883.626,A -85,B 0,C 180,E1 7259.222,E2 7259.222} C_VEL
LIN {X 0,Y 209.088,Z 867.493,A -85,B 0,C 180,E1 7255.973,E2 7255.973} C_VEL
LIN {X 0,Y 219.509,Z 850.614,A -85,B 0,C 180,E1 7253.36,E2 7253.36} C_VEL
LIN {X 0,Y 229.127,Z 832.847,A -85,B 0,C 180,E1 7251.224,E2 7251.224} C_VEL
LIN {X 0,Y 238.17,Z 813.28,A -85,B 0,C 180,E1 7249.4,E2 7249.4} C_VEL
LIN {X 0,Y 245.748,Z 793.579,A -85,B 0,C 180,E1 7247.983,E2 7247.983} C_VEL
LIN {X 0,Y 252.146,Z 773.184,A -85,B 0,C 180,E1 7246.857,E2 7246.857} C_VEL
LIN {X 0,Y 257.542,Z 750.903,A -85,B 0,C 180,E1 7245.944,E2 7245.944} C_VEL
LIN {X 0,Y 261.346,Z 728.565,A -85,B 0,C 180,E1 7245.308,E2 7245.308} C_VEL
LIN {X 0,Y 274.672,Z 607.232,A -85,B 0,C 180,E1 7242.829,E2 7242.829} C_VEL
LIN {X 0,Y 269.934,Z 597.548,A -85,B 0,C 180,E1 7239.028,E2 7239.028} C_VEL
LIN {X 0,Y 266.314,Z 590.84,A -85,B 0,C 180,E1 7235.588,E2 7235.588} C_VEL
LIN {X 0,Y 263.862,Z 586.429,A -85,B 0,C 180,E1 7232.812,E2 7232.812} C_VEL
LIN {X 0,Y 262.132,Z 583.291,A -85,B 0,C 180,E1 7230.485,E2 7230.485} C_VEL
LIN {X 0,Y 260.202,Z 579.759,A -85,B 0,C 180,E1 7227.212,E2 7227.212} C_VEL
LIN {X 0,Y 258.19,Z 576.027,A -85,B 0,C 180,E1 7221.648,E2 7221.648} C_VEL
LIN {X 0,Y 257.6,Z 575.401,A -85,B 0,C 180,E1 7216.229,E2 7216.229} C_VEL
LIN {X 0,Y 258.482,Z 576.395,A -85,B 0,C 180,E1 7211.153,E2 7211.153} C_VEL
LIN {X 0,Y 261.047,Z 580.91,A -85,B 0,C 180,E1 7205.191,E2 7205.191} C_VEL
LIN {X 0,Y 263.717,Z 585.575,A -85,B 0,C 180,E1 7201.304,E2 7201.304} C_VEL
LIN {X 0,Y 266.452,Z 590.416,A -85,B 0,C 180,E1 7198.173,E2 7198.173} C_VEL
LIN {X 0,Y 269.98,Z 596.63,A -85,B 0,C 180,E1 7194.843,E2 7194.843} C_VEL
LIN {X 0,Y 275.378,Z 606.867,A -85,B 0,C 180,E1 7190.597,E2 7190.597} C_VEL
LIN {X 0,Y 277.987,Z 612.275,A -85,B 0,C 180,E1 7188.783,E2 7188.783} C_VEL
LIN {X 0,Y 269.949,Z 690.264,A -85,B 0,C 180,E1 7187.236,E2 7187.236} C_VEL
LIN {X 0,Y 268.787,Z 697.936,A -85,B 0,C 180,E1 7187.269,E2 7187.269} C_VEL
LIN {X 0,Y 264.24,Z 718.331,A -85,B 0,C 180,E1 7188.104,E2 7188.104} C_VEL
LIN {X 0,Y 263.258,Z 724.92,A -85,B 0,C 180,E1 7188.127,E2 7188.127} C_VEL
LIN {X 0,Y 259.92,Z 750.89,A -85,B 0,C 180,E1 7187.55,E2 7187.55} C_VEL
LIN {X 0,Y 255.349,Z 772.956,A -85,B 0,C 180,E1 7186.924,E2 7186.924} C_VEL
LIN {X 0,Y 249.479,Z 793.78,A -85,B 0,C 180,E1 7186.154,E2 7186.154} C_VEL
LIN {X 0,Y 242.122,Z 814.368,A -85,B 0,C 180,E1 7185.1,E2 7185.1} C_VEL
LIN {X 0,Y 233.813,Z 833.688,A -85,B 0,C 180,E1 7183.788,E2 7183.788} C_VEL
LIN {X 0,Y 223.883,Z 853.341,A -85,B 0,C 180,E1 7182.049,E2 7182.049} C_VEL
LIN {X 0,Y 213.446,Z 871.288,A -85,B 0,C 180,E1 7179.974,E2 7179.974} C_VEL
LIN {X 0,Y 202.038,Z 888.47,A -85,B 0,C 180,E1 7177.375,E2 7177.375} C_VEL
LIN {X 0,Y 190.401,Z 904.103,A -85,B 0,C 180,E1 7174.248,E2 7174.248} C_VEL
LIN {X 0,Y 178.326,Z 918.818,A -85,B 0,C 180,E1 7170.362,E2 7170.362} C_VEL
LIN {X 0,Y 166.861,Z 931.758,A -85,B 0,C 180,E1 7165.794,E2 7165.794} C_VEL
LIN {X 0,Y 155.439,Z 943.922,A -85,B 0,C 180,E1 7159.958,E2 7159.958} C_VEL
LIN {X 0,Y 145.767,Z 953.914,A -85,B 0,C 180,E1 7153.319,E2 7153.319} C_VEL
LIN {X 0,Y 137.791,Z 962.464,A -85,B 0,C 180,E1 7145.496,E2 7145.496} C_VEL
LIN {X 0,Y 132.29,Z 969.207,A -85,B 0,C 180,E1 7136.895,E2 7136.895} C_VEL
LIN {X 0,Y 129.408,Z 974.084,A -85,B 0,C 180,E1 7128.012,E2 7128.012} C_VEL
LIN {X 0,Y 128.736,Z 977.127,A -85,B 0,C 180,E1 7119.396,E2 7119.396} C_VEL
LIN {X 0,Y 129.015,Z 978.409,A -85,B 0,C 180,E1 7113.119,E2 7113.119} C_VEL
LIN {X 0,Y 129.046,Z 978.788,A -85,B 0,C 180,E1 7108.145,E2 7108.145} C_VEL
LIN {X 0,Y 128.7,Z 978.478,A -85,B 0,C 180,E1 7101.971,E2 7101.971} C_VEL
LIN {X 0,Y 129.073,Z 976.884,A -85,B 0,C 180,E1 7093.355,E2 7093.355} C_VEL
LIN {X 0,Y 131.849,Z 973.448,A -85,B 0,C 180,E1 7083.918,E2 7083.918} C_VEL
LIN {X 0,Y 138.179,Z 967.916,A -85,B 0,C 180,E1 7074.131,E2 7074.131} C_VEL
LIN {X 0,Y 147.397,Z 960.809,A -85,B 0,C 180,E1 7065.691,E2 7065.691} C_VEL
LIN {X 0,Y 159.041,Z 952.022,A -85,B 0,C 180,E1 7058.49,E2 7058.49} C_VEL
LIN {X 0,Y 172.116,Z 941.776,A -85,B 0,C 180,E1 7052.629,E2 7052.629} C_VEL
LIN {X 0,Y 186.413,Z 929.905,A -85,B 0,C 180,E1 7047.765,E2 7047.765} C_VEL
LIN {X 0,Y 201.123,Z 916.667,A -85,B 0,C 180,E1 7043.851,E2 7043.851} C_VEL
LIN {X 0,Y 215.857,Z 902.073,A -85,B 0,C 180,E1 7040.684,E2 7040.684} C_VEL
LIN {X 0,Y 230.363,Z 885.929,A -85,B 0,C 180,E1 7038.119,E2 7038.119} C_VEL
LIN {X 0,Y 243.992,Z 868.786,A -85,B 0,C 180,E1 7036.087,E2 7036.087} C_VEL
LIN {X 0,Y 256.592,Z 850.816,A -85,B 0,C 180,E1 7034.485,E2 7034.485} C_VEL
LIN {X 0,Y 267.575,Z 832.788,A -85,B 0,C 180,E1 7033.267,E2 7033.267} C_VEL
LIN {X 0,Y 277.618,Z 813.368,A -85,B 0,C 180,E1 7032.282,E2 7032.282} C_VEL
LIN {X 0,Y 286.211,Z 793.457,A -85,B 0,C 180,E1 7031.535,E2 7031.535} C_VEL
LIN {X 0,Y 292.632,Z 775.475,A -85,B 0,C 180,E1 7031.014,E2 7031.014} C_VEL
LIN {X 0,Y 285.213,Z 795.488,A -85,B 0,C 180,E1 7030.229,E2 7030.229} C_VEL
LIN {X 0,Y 276.536,Z 814.485,A -85,B 0,C 180,E1 7029.262,E2 7029.262} C_VEL
LIN {X 0,Y 266.571,Z 832.757,A -85,B 0,C 180,E1 7028.067,E2 7028.067} C_VEL
LIN {X 0,Y 255.646,Z 849.876,A -85,B 0,C 180,E1 7026.634,E2 7026.634} C_VEL
LIN {X 0,Y 243.304,Z 866.453,A -85,B 0,C 180,E1 7024.841,E2 7024.841} C_VEL
LIN {X 0,Y 230.187,Z 881.915,A -85,B 0,C 180,E1 7022.66,E2 7022.66} C_VEL
LIN {X 0,Y 216.385,Z 896.22,A -85,B 0,C 180,E1 7019.999,E2 7019.999} C_VEL
LIN {X 0,Y 202.266,Z 909.201,A -85,B 0,C 180,E1 7016.763,E2 7016.763} C_VEL
LIN {X 0,Y 187.494,Z 921.185,A -85,B 0,C 180,E1 7012.633,E2 7012.633} C_VEL
LIN {X 0,Y 173.852,Z 931.06,A -85,B 0,C 180,E1 7007.837,E2 7007.837} C_VEL
LIN {X 0,Y 160.815,Z 939.618,A -85,B 0,C 180,E1 7001.887,E2 7001.887} C_VEL
LIN {X 0,Y 149.272,Z 946.514,A -85,B 0,C 180,E1 6994.701,E2 6994.701} C_VEL
LIN {X 0,Y 140.404,Z 951.401,A -85,B 0,C 180,E1 6986.745,E2 6986.745} C_VEL
LIN {X 0,Y 133.972,Z 954.671,A -85,B 0,C 180,E1 6977.619,E2 6977.619} C_VEL
LIN {X 0,Y 130.598,Z 956.029,A -85,B 0,C 180,E1 6968.654,E2 6968.654} C_VEL
LIN {X 0,Y 129.366,Z 955.999,A -85,B 0,C 180,E1 6960.042,E2 6960.042} C_VEL
LIN {X 0,Y 129.359,Z 954.883,A -85,B 0,C 180,E1 6952.245,E2 6952.245} C_VEL
LIN {X 0,Y 130.653,Z 952.32,A -85,B 0,C 180,E1 6943.608,E2 6943.608} C_VEL
LIN {X 0,Y 133.825,Z 948.332,A -85,B 0,C 180,E1 6935.135,E2 6935.135} C_VEL
LIN {X 0,Y 139.473,Z 942.412,A -85,B 0,C 180,E1 6926.704,E2 6926.704} C_VEL
LIN {X 0,Y 147.355,Z 934.627,A -85,B 0,C 180,E1 6919.04,E2 6919.04} C_VEL
LIN {X 0,Y 156.688,Z 925.402,A -85,B 0,C 180,E1 6912.54,E2 6912.54} C_VEL
LIN {X 0,Y 167.568,Z 914.198,A -85,B 0,C 180,E1 6906.801,E2 6906.801} C_VEL
LIN {X 0,Y 178.621,Z 901.992,A -85,B 0,C 180,E1 6902.184,E2 6902.184} C_VEL
LIN {X 0,Y 190.082,Z 888.17,A -85,B 0,C 180,E1 6898.257,E2 6898.257} C_VEL
LIN {X 0,Y 201.741,Z 872.468,A -85,B 0,C 180,E1 6894.9,E2 6894.9} C_VEL
LIN {X 0,Y 212.604,Z 855.881,A -85,B 0,C 180,E1 6892.195,E2 6892.195} C_VEL
LIN {X 0,Y 222.542,Z 838.605,A -85,B 0,C 180,E1 6890.017,E2 6890.017} C_VEL
LIN {X 0,Y 232.161,Z 819.188,A -85,B 0,C 180,E1 6888.117,E2 6888.117} C_VEL
LIN {X 0,Y 240.314,Z 799.648,A -85,B 0,C 180,E1 6886.641,E2 6886.641} C_VEL
LIN {X 0,Y 247.317,Z 779.208,A -85,B 0,C 180,E1 6885.453,E2 6885.453} C_VEL
LIN {X 0,Y 253.1,Z 757.609,A -85,B 0,C 180,E1 6884.519,E2 6884.519} C_VEL
LIN {X 0,Y 257.319,Z 735.815,A -85,B 0,C 180,E1 6883.845,E2 6883.845} C_VEL
LIN {X 0,Y 261.536,Z 701.244,A -85,B 0,C 180,E1 6883.112,E2 6883.112} C_VEL
LIN {X 0,Y 271.417,Z 611.919,A -85,B 0,C 180,E1 6881.326,E2 6881.326} C_VEL
LIN {X 0,Y 266.893,Z 602.531,A -85,B 0,C 180,E1 6877.366,E2 6877.366} C_VEL
LIN {X 0,Y 263.219,Z 595.479,A -85,B 0,C 180,E1 6873.422,E2 6873.422} C_VEL
LIN {X 0,Y 260.711,Z 590.904,A -85,B 0,C 180,E1 6870.033,E2 6870.033} C_VEL
LIN {X 0,Y 258.924,Z 587.512,A -85,B 0,C 180,E1 6866.86,E2 6866.86} C_VEL
LIN {X 0,Y 257.067,Z 583.912,A -85,B 0,C 180,E1 6861.446,E2 6861.446} C_VEL
LIN {X 0,Y 256.55,Z 583.334,A -85,B 0,C 180,E1 6855.832,E2 6855.832} C_VEL
LIN {X 0,Y 257.382,Z 584.387,A -85,B 0,C 180,E1 6851.201,E2 6851.201} C_VEL
LIN {X 0,Y 259.754,Z 588.67,A -85,B 0,C 180,E1 6845.523,E2 6845.523} C_VEL
LIN {X 0,Y 262.245,Z 593.173,A -85,B 0,C 180,E1 6841.749,E2 6841.749} C_VEL
LIN {X 0,Y 265.006,Z 598.224,A -85,B 0,C 180,E1 6838.487,E2 6838.487} C_VEL
LIN {X 0,Y 268.402,Z 604.433,A -85,B 0,C 180,E1 6835.193,E2 6835.193} C_VEL
LIN {X 0,Y 273.354,Z 614.171,A -85,B 0,C 180,E1 6831.164,E2 6831.164} C_VEL
LIN {X 0,Y 274.599,Z 616.941,A -85,B 0,C 180,E1 6830.242,E2 6830.242} C_VEL
LIN {X 0,Y 263.258,Z 724.92,A -85,B 0,C 180,E1 6828.127,E2 6828.127} C_VEL
LIN {X 0,Y 262.064,Z 732.592,A -85,B 0,C 180,E1 6828.181,E2 6828.181} C_VEL
LIN {X 0,Y 256.789,Z 752.857,A -85,B 0,C 180,E1 6828.985,E2 6828.985} C_VEL
LIN {X 0,Y 255.231,Z 759.333,A -85,B 0,C 180,E1 6828.967,E2 6828.967} C_VEL
LIN {X 0,Y 249.917,Z 781.33,A -85,B 0,C 180,E1 6828.305,E2 6828.305} C_VEL
LIN {X 0,Y 243.287,Z 801.985,A -85,B 0,C 180,E1 6827.456,E2 6827.456} C_VEL
LIN {X 0,Y 235.609,Z 821.518,A -85,B 0,C 180,E1 6826.378,E2 6826.378} C_VEL
LIN {X 0,Y 226.712,Z 840.637,A -85,B 0,C 180,E1 6824.996,E2 6824.996} C_VEL
LIN {X 0,Y 216.673,Z 859.124,A -85,B 0,C 180,E1 6823.255,E2 6823.255} C_VEL
LIN {X 0,Y 205.602,Z 876.706,A -85,B 0,C 180,E1 6821.075,E2 6821.075} C_VEL
LIN {X 0,Y 193.661,Z 893.476,A -85,B 0,C 180,E1 6818.343,E2 6818.343} C_VEL
LIN {X 0,Y 181.845,Z 908.387,A -85,B 0,C 180,E1 6815.138,E2 6815.138} C_VEL
LIN {X 0,Y 169.236,Z 922.84,A -85,B 0,C 180,E1 6810.985,E2 6810.985} C_VEL
LIN {X 0,Y 156.99,Z 935.688,A -85,B 0,C 180,E1 6805.901,E2 6805.901} C_VEL
LIN {X 0,Y 145.896,Z 946.704,A -85,B 0,C 180,E1 6799.896,E2 6799.896} C_VEL
LIN {X 0,Y 135.566,Z 956.821,A -85,B 0,C 180,E1 6792.168,E2 6792.168} C_VEL
LIN {X 0,Y 128.003,Z 964.653,A -85,B 0,C 180,E1 6783.693,E2 6783.693} C_VEL
LIN {X 0,Y 123.137,Z 970.632,A -85,B 0,C 180,E1 6774.474,E2 6774.474} C_VEL
LIN {X 0,Y 121.026,Z 974.647,A -85,B 0,C 180,E1 6765.339,E2 6765.339} C_VEL
LIN {X 0,Y 120.845,Z 977.073,A -85,B 0,C 180,E1 6756.858,E2 6756.858} C_VEL
LIN {X 0,Y 121.131,Z 977.988,A -85,B 0,C 180,E1 6750.483,E2 6750.483} C_VEL
LIN {X 0,Y 120.848,Z 978.048,A -85,B 0,C 180,E1 6744.312,E2 6744.312} C_VEL
LIN {X 0,Y 120.831,Z 976.881,A -85,B 0,C 180,E1 6735.497,E2 6735.497} C_VEL
LIN {X 0,Y 123.042,Z 974.183,A -85,B 0,C 180,E1 6725.52,E2 6725.52} C_VEL
LIN {X 0,Y 128.647,Z 969.524,A -85,B 0,C 180,E1 6715.446,E2 6715.446} C_VEL
LIN {X 0,Y 137.56,Z 963.143,A -85,B 0,C 180,E1 6706.343,E2 6706.343} C_VEL
LIN {X 0,Y 149.382,Z 954.951,A -85,B 0,C 180,E1 6698.469,E2 6698.469} C_VEL
LIN {X 0,Y 162.89,Z 945.324,A -85,B 0,C 180,E1 6692.122,E2 6692.122} C_VEL
LIN {X 0,Y 177.353,Z 934.244,A -85,B 0,C 180,E1 6687.051,E2 6687.051} C_VEL
LIN {X 0,Y 193.048,Z 921.2,A -85,B 0,C 180,E1 6682.812,E2 6682.812} C_VEL
LIN {X 0,Y 208.849,Z 906.65,A -85,B 0,C 180,E1 6679.438,E2 6679.438} C_VEL
LIN {X 0,Y 223.366,Z 891.781,A -85,B 0,C 180,E1 6676.915,E2 6676.915} C_VEL
LIN {X 0,Y 237.182,Z 875.769,A -85,B 0,C 180,E1 6674.9,E2 6674.9} C_VEL
LIN {X 0,Y 250.13,Z 858.727,A -85,B 0,C 180,E1 6673.285,E2 6673.285} C_VEL
LIN {X 0,Y 262.157,Z 840.709,A -85,B 0,C 180,E1 6671.994,E2 6671.994} C_VEL
LIN {X 0,Y 272.848,Z 822.012,A -85,B 0,C 180,E1 6670.985,E2 6670.985} C_VEL
LIN {X 0,Y 274.936,Z 817.879,A -85,B 0,C 180,E1 6670.783,E2 6670.783} C_VEL
LIN {X 0,Y 264.207,Z 836.589,A -85,B 0,C 180,E1 6669.584,E2 6669.584} C_VEL
LIN {X 0,Y 252.48,Z 853.965,A -85,B 0,C 180,E1 6668.142,E2 6668.142} C_VEL
LIN {X 0,Y 240.208,Z 869.774,A -85,B 0,C 180,E1 6666.452,E2 6666.452} C_VEL
LIN {X 0,Y 226.475,Z 885.056,A -85,B 0,C 180,E1 6664.304,E2 6664.304} C_VEL
LIN {X 0,Y 211.848,Z 899.393,A -85,B 0,C 180,E1 6661.622,E2 6661.622} C_VEL
LIN {X 0,Y 196.551,Z 912.563,A -85,B 0,C 180,E1 6658.25,E2 6658.25} C_VEL
LIN {X 0,Y 182.055,Z 923.632,A -85,B 0,C 180,E1 6654.326,E2 6654.326} C_VEL
LIN {X 0,Y 167.462,Z 933.549,A -85,B 0,C 180,E1 6649.333,E2 6649.333} C_VEL
LIN {X 0,Y 154.235,Z 941.51,A -85,B 0,C 180,E1 6643.426,E2 6643.426} C_VEL
LIN {X 0,Y 142.759,Z 947.77,A -85,B 0,C 180,E1 6636.469,E2 6636.469} C_VEL
LIN {X 0,Y 132.788,Z 952.706,A -85,B 0,C 180,E1 6627.681,E2 6627.681} C_VEL
LIN {X 0,Y 126.392,Z 955.567,A -85,B 0,C 180,E1 6618.706,E2 6618.706} C_VEL
LIN {X 0,Y 122.749,Z 956.836,A -85,B 0,C 180,E1 6609.299,E2 6609.299} C_VEL
LIN {X 0,Y 121.399,Z 956.687,A -85,B 0,C 180,E1 6600.138,E2 6600.138} C_VEL
LIN {X 0,Y 121.418,Z 955.5,A -85,B 0,C 180,E1 6591.739,E2 6591.739} C_VEL
LIN {X 0,Y 122.872,Z 952.864,A -85,B 0,C 180,E1 6582.681,E2 6582.681} C_VEL
LIN {X 0,Y 126.698,Z 948.451,A -85,B 0,C 180,E1 6573.157,E2 6573.157} C_VEL
LIN {X 0,Y 132.655,Z 942.719,A -85,B 0,C 180,E1 6564.802,E2 6564.802} C_VEL
LIN {X 0,Y 141.186,Z 934.835,A -85,B 0,C 180,E1 6556.893,E2 6556.893} C_VEL
LIN {X 0,Y 151.156,Z 925.481,A -85,B 0,C 180,E1 6550.277,E2 6550.277} C_VEL
LIN {X 0,Y 162.021,Z 914.784,A -85,B 0,C 180,E1 6544.791,E2 6544.791} C_VEL
LIN {X 0,Y 173.32,Z 902.823,A -85,B 0,C 180,E1 6540.249,E2 6540.249} C_VEL
LIN {X 0,Y 185.457,Z 888.701,A -85,B 0,C 180,E1 6536.262,E2 6536.262} C_VEL
LIN {X 0,Y 197.505,Z 872.97,A -85,B 0,C 180,E1 6532.949,E2 6532.949} C_VEL
LIN {X 0,Y 208.436,Z 856.742,A -85,B 0,C 180,E1 6530.351,E2 6530.351} C_VEL
LIN {X 0,Y 218.897,Z 839.031,A -85,B 0,C 180,E1 6528.167,E2 6528.167} C_VEL
LIN {X 0,Y 228.753,Z 819.577,A -85,B 0,C 180,E1 6526.317,E2 6526.317} C_VEL
LIN {X 0,Y 237.093,Z 800.006,A -85,B 0,C 180,E1 6524.883,E2 6524.883} C_VEL
LIN {X 0,Y 244.039,Z 780.243,A -85,B 0,C 180,E1 6523.765,E2 6523.765} C_VEL
LIN {X 0,Y 249.986,Z 758.556,A -85,B 0,C 180,E1 6522.851,E2 6522.851} C_VEL
LIN {X 0,Y 254.27,Z 737.119,A -85,B 0,C 180,E1 6522.2,E2 6522.2} C_VEL
LIN {X 0,Y 258.244,Z 706.022,A -85,B 0,C 180,E1 6521.548,E2 6521.548} C_VEL
LIN {X 0,Y 268.336,Z 616.78,A -85,B 0,C 180,E1 6519.797,E2 6519.797} C_VEL
LIN {X 0,Y 264.782,Z 609.211,A -85,B 0,C 180,E1 6516.45,E2 6516.45} C_VEL
LIN {X 0,Y 261.353,Z 602.448,A -85,B 0,C 180,E1 6512.515,E2 6512.515} C_VEL
LIN {X 0,Y 259.376,Z 598.64,A -85,B 0,C 180,E1 6509.694,E2 6509.694} C_VEL
LIN {X 0,Y 257.652,Z 595.265,A -85,B 0,C 180,E1 6506.506,E2 6506.506} C_VEL
LIN {X 0,Y 255.952,Z 591.812,A -85,B 0,C 180,E1 6501.304,E2 6501.304} C_VEL
LIN {X 0,Y 255.472,Z 591.261,A -85,B 0,C 180,E1 6495.901,E2 6495.901} C_VEL
LIN {X 0,Y 256.222,Z 592.203,A -85,B 0,C 180,E1 6491.48,E2 6491.48} C_VEL
LIN {X 0,Y 258.514,Z 596.535,A -85,B 0,C 180,E1 6485.772,E2 6485.772} C_VEL
LIN {X 0,Y 260.87,Z 600.937,A -85,B 0,C 180,E1 6482.087,E2 6482.087} C_VEL
LIN {X 0,Y 263.473,Z 605.842,A -85,B 0,C 180,E1 6478.913,E2 6478.913} C_VEL
LIN {X 0,Y 266.825,Z 612.21,A -85,B 0,C 180,E1 6475.554,E2 6475.554} C_VEL
LIN {X 0,Y 271.355,Z 621.511,A -85,B 0,C 180,E1 6471.735,E2 6471.735} C_VEL
LIN {X 0,Y 257.864,Z 744.547,A -85,B 0,C 180,E1 6469.342,E2 6469.342} C_VEL
LIN {X 0,Y 255.231,Z 759.333,A -85,B 0,C 180,E1 6468.967,E2 6468.967} C_VEL
LIN {X 0,Y 253.206,Z 766.825,A -85,B 0,C 180,E1 6468.986,E2 6468.986} C_VEL
LIN {X 0,Y 245.58,Z 786.434,A -85,B 0,C 180,E1 6469.67,E2 6469.67} C_VEL
LIN {X 0,Y 243.29,Z 792.679,A -85,B 0,C 180,E1 6469.596,E2 6469.596} C_VEL
LIN {X 0,Y 235.613,Z 813.458,A -85,B 0,C 180,E1 6468.62,E2 6468.62} C_VEL
LIN {X 0,Y 226.948,Z 832.846,A -85,B 0,C 180,E1 6467.4,E2 6467.4} C_VEL
LIN {X 0,Y 216.619,Z 852.439,A -85,B 0,C 180,E1 6465.783,E2 6465.783} C_VEL
LIN {X 0,Y 205.689,Z 870.362,A -85,B 0,C 180,E1 6463.834,E2 6463.834} C_VEL
LIN {X 0,Y 193.39,Z 887.924,A -85,B 0,C 180,E1 6461.305,E2 6461.305} C_VEL
LIN {X 0,Y 180.877,Z 903.677,A -85,B 0,C 180,E1 6458.243,E2 6458.243} C_VEL
LIN {X 0,Y 168.333,Z 917.878,A -85,B 0,C 180,E1 6454.548,E2 6454.548} C_VEL
LIN {X 0,Y 155.807,Z 930.859,A -85,B 0,C 180,E1 6449.965,E2 6449.965} C_VEL
LIN {X 0,Y 143.645,Z 942.61,A -85,B 0,C 180,E1 6444.22,E2 6444.22} C_VEL
LIN {X 0,Y 132.479,Z 952.879,A -85,B 0,C 180,E1 6437.073,E2 6437.073} C_VEL
LIN {X 0,Y 123.766,Z 960.987,A -85,B 0,C 180,E1 6429.071,E2 6429.071} C_VEL
LIN {X 0,Y 117.187,Z 967.794,A -85,B 0,C 180,E1 6419.512,E2 6419.512} C_VEL
LIN {X 0,Y 113.682,Z 972.652,A -85,B 0,C 180,E1 6409.536,E2 6409.536} C_VEL
LIN {X 0,Y 112.788,Z 975.698,A -85,B 0,C 180,E1 6399.707,E2 6399.707} C_VEL
LIN {X 0,Y 113.107,Z 976.968,A -85,B 0,C 180,E1 6392.544,E2 6392.544} C_VEL
LIN {X 0,Y 113.077,Z 977.306,A -85,B 0,C 180,E1 6387.477,E2 6387.477} C_VEL
LIN {X 0,Y 112.697,Z 977,A -85,B 0,C 180,E1 6380.307,E2 6380.307} C_VEL
LIN {X 0,Y 113.577,Z 975.408,A -85,B 0,C 180,E1 6370.378,E2 6370.378} C_VEL
LIN {X 0,Y 117.718,Z 971.864,A -85,B 0,C 180,E1 6359.375,E2 6359.375} C_VEL
LIN {X 0,Y 125.922,Z 966.348,A -85,B 0,C 180,E1 6348.788,E2 6348.788} C_VEL
LIN {X 0,Y 137.092,Z 959.298,A -85,B 0,C 180,E1 6340.038,E2 6340.038} C_VEL
LIN {X 0,Y 150.918,Z 950.374,A -85,B 0,C 180,E1 6332.73,E2 6332.73} C_VEL
LIN {X 0,Y 166.032,Z 939.894,A -85,B 0,C 180,E1 6326.987,E2 6326.987} C_VEL
LIN {X 0,Y 181.768,Z 928.06,A -85,B 0,C 180,E1 6322.485,E2 6322.485} C_VEL
LIN {X 0,Y 198.115,Z 914.475,A -85,B 0,C 180,E1 6318.843,E2 6318.843} C_VEL
LIN {X 0,Y 214.122,Z 899.582,A -85,B 0,C 180,E1 6315.991,E2 6315.991} C_VEL
LIN {X 0,Y 229.065,Z 883.832,A -85,B 0,C 180,E1 6313.814,E2 6313.814} C_VEL
LIN {X 0,Y 243.314,Z 866.761,A -85,B 0,C 180,E1 6312.067,E2 6312.067} C_VEL
LIN {X 0,Y 256.76,Z 848.214,A -85,B 0,C 180,E1 6310.668,E2 6310.668} C_VEL
LIN {X 0,Y 257.331,Z 847.358,A -85,B 0,C 180,E1 6310.606,E2 6310.606} C_VEL
LIN {X 0,Y 244.486,Z 864.444,A -85,B 0,C 180,E1 6309.059,E2 6309.059} C_VEL
LIN {X 0,Y 230.749,Z 880.244,A -85,B 0,C 180,E1 6307.182,E2 6307.182} C_VEL
LIN {X 0,Y 216.226,Z 894.731,A -85,B 0,C 180,E1 6304.884,E2 6304.884} C_VEL
LIN {X 0,Y 200.846,Z 908.163,A -85,B 0,C 180,E1 6301.996,E2 6301.996} C_VEL
LIN {X 0,Y 185.021,Z 920.292,A -85,B 0,C 180,E1 6298.37,E2 6298.37} C_VEL
LIN {X 0,Y 169.879,Z 930.559,A -85,B 0,C 180,E1 6294.005,E2 6294.005} C_VEL
LIN {X 0,Y 155.001,Z 939.474,A -85,B 0,C 180,E1 6288.464,E2 6288.464} C_VEL
LIN {X 0,Y 141.244,Z 946.742,A -85,B 0,C 180,E1 6281.513,E2 6281.513} C_VEL
LIN {X 0,Y 129.826,Z 952.059,A -85,B 0,C 180,E1 6273.276,E2 6273.276} C_VEL
LIN {X 0,Y 121.315,Z 955.554,A -85,B 0,C 180,E1 6263.852,E2 6263.852} C_VEL
LIN {X 0,Y 115.802,Z 957.409,A -85,B 0,C 180,E1 6252.992,E2 6252.992} C_VEL
LIN {X 0,Y 113.666,Z 957.617,A -85,B 0,C 180,E1 6243.037,E2 6243.037} C_VEL
LIN {X 0,Y 113.314,Z 956.656,A -85,B 0,C 180,E1 6234.489,E2 6234.489} C_VEL
LIN {X 0,Y 114.285,Z 954.608,A -85,B 0,C 180,E1 6225.205,E2 6225.205} C_VEL
LIN {X 0,Y 117.473,Z 950.778,A -85,B 0,C 180,E1 6215.219,E2 6215.219} C_VEL
LIN {X 0,Y 123.317,Z 945.281,A -85,B 0,C 180,E1 6205.799,E2 6205.799} C_VEL
LIN {X 0,Y 131.737,Z 937.962,A -85,B 0,C 180,E1 6197.276,E2 6197.276} C_VEL
LIN {X 0,Y 141.757,Z 929.236,A -85,B 0,C 180,E1 6190.202,E2 6190.202} C_VEL
LIN {X 0,Y 153.399,Z 918.56,A -85,B 0,C 180,E1 6184.098,E2 6184.098} C_VEL
LIN {X 0,Y 165.622,Z 906.349,A -85,B 0,C 180,E1 6179.119,E2 6179.119} C_VEL
LIN {X 0,Y 177.279,Z 893.55,A -85,B 0,C 180,E1 6175.268,E2 6175.268} C_VEL
LIN {X 0,Y 189.948,Z 878.071,A -85,B 0,C 180,E1 6171.786,E2 6171.786} C_VEL
LIN {X 0,Y 201.511,Z 862.093,A -85,B 0,C 180,E1 6169.077,E2 6169.077} C_VEL
LIN {X 0,Y 212.529,Z 844.703,A -85,B 0,C 180,E1 6166.821,E2 6166.821} C_VEL
LIN {X 0,Y 222.816,Z 825.719,A -85,B 0,C 180,E1 6164.939,E2 6164.939} C_VEL
LIN {X 0,Y 231.53,Z 806.647,A -85,B 0,C 180,E1 6163.483,E2 6163.483} C_VEL
LIN {X 0,Y 239.236,Z 786.27,A -85,B 0,C 180,E1 6162.284,E2 6162.284} C_VEL
LIN {X 0,Y 245.837,Z 764.229,A -85,B 0,C 180,E1 6161.315,E2 6161.315} C_VEL
LIN {X 0,Y 250.682,Z 742.497,A -85,B 0,C 180,E1 6160.623,E2 6160.623} C_VEL
LIN {X 0,Y 254.052,Z 719.961,A -85,B 0,C 180,E1 6160.121,E2 6160.121} C_VEL
LIN {X 0,Y 265.395,Z 621.791,A -85,B 0,C 180,E1 6158.267,E2 6158.267} C_VEL
LIN {X 0,Y 262.05,Z 614.426,A -85,B 0,C 180,E1 6154.78,E2 6154.78} C_VEL
LIN {X 0,Y 259.177,Z 608.714,A -85,B 0,C 180,E1 6151.129,E2 6151.129} C_VEL
LIN {X 0,Y 257.777,Z 605.876,A -85,B 0,C 180,E1 6148.876,E2 6148.876} C_VEL
LIN {X 0,Y 256.39,Z 603.018,A -85,B 0,C 180,E1 6146.147,E2 6146.147} C_VEL
LIN {X 0,Y 254.837,Z 599.712,A -85,B 0,C 180,E1 6141.16,E2 6141.16} C_VEL
LIN {X 0,Y 254.416,Z 599.199,A -85,B 0,C 180,E1 6135.655,E2 6135.655} C_VEL
LIN {X 0,Y 255.123,Z 600.2,A -85,B 0,C 180,E1 6131.526,E2 6131.526} C_VEL
LIN {X 0,Y 257.225,Z 604.262,A -85,B 0,C 180,E1 6126.137,E2 6126.137} C_VEL
LIN {X 0,Y 259.504,Z 608.699,A -85,B 0,C 180,E1 6122.43,E2 6122.43} C_VEL
LIN {X 0,Y 262.138,Z 613.82,A -85,B 0,C 180,E1 6119.126,E2 6119.126} C_VEL
LIN {X 0,Y 265.671,Z 620.844,A -85,B 0,C 180,E1 6115.522,E2 6115.522} C_VEL
LIN {X 0,Y 268.208,Z 626.549,A -85,B 0,C 180,E1 6113.251,E2 6113.251} C_VEL
LIN {X 0,Y 255.04,Z 743.978,A -85,B 0,C 180,E1 6111.021,E2 6111.021} C_VEL
LIN {X 0,Y 250.728,Z 766.236,A -85,B 0,C 180,E1 6110.459,E2 6110.459} C_VEL
LIN {X 0,Y 244.864,Z 787.628,A -85,B 0,C 180,E1 6109.78,E2 6109.78} C_VEL
LIN {X 0,Y 243.29,Z 792.679,A -85,B 0,C 180,E1 6109.596,E2 6109.596} C_VEL
LIN {X 0,Y 240.38,Z 799.943,A -85,B 0,C 180,E1 6109.506,E2 6109.506} C_VEL
LIN {X 0,Y 231.025,Z 817.782,A -85,B 0,C 180,E1 6109.961,E2 6109.961} C_VEL
LIN {X 0,Y 227.619,Z 824.521,A -85,B 0,C 180,E1 6109.793,E2 6109.793} C_VEL
LIN {X 0,Y 217.911,Z 843.815,A -85,B 0,C 180,E1 6108.431,E2 6108.431} C_VEL
LIN {X 0,Y 206.583,Z 863.029,A -85,B 0,C 180,E1 6106.633,E2 6106.633} C_VEL
LIN {X 0,Y 194.609,Z 880.595,A -85,B 0,C 180,E1 6104.453,E2 6104.453} C_VEL
LIN {X 0,Y 182.047,Z 896.836,A -85,B 0,C 180,E1 6101.757,E2 6101.757} C_VEL
LIN {X 0,Y 168.888,Z 911.847,A -85,B 0,C 180,E1 6098.368,E2 6098.368} C_VEL
LIN {X 0,Y 155.591,Z 925.541,A -85,B 0,C 180,E1 6094.129,E2 6094.129} C_VEL
LIN {X 0,Y 141.895,Z 938.43,A -85,B 0,C 180,E1 6088.512,E2 6088.512} C_VEL
LIN {X 0,Y 130.28,Z 948.72,A -85,B 0,C 180,E1 6082.124,E2 6082.124} C_VEL
LIN {X 0,Y 119.672,Z 957.885,A -85,B 0,C 180,E1 6073.917,E2 6073.917} C_VEL
LIN {X 0,Y 111.655,Z 965.121,A -85,B 0,C 180,E1 6064.356,E2 6064.356} C_VEL
LIN {X 0,Y 106.556,Z 970.808,A -85,B 0,C 180,E1 6053.222,E2 6053.222} C_VEL
LIN {X 0,Y 104.857,Z 974.371,A -85,B 0,C 180,E1 6042.68,E2 6042.68} C_VEL
LIN {X 0,Y 105.073,Z 976.053,A -85,B 0,C 180,E1 6033.831,E2 6033.831} C_VEL
LIN {X 0,Y 105.153,Z 976.553,A -85,B 0,C 180,E1 6028.377,E2 6028.377} C_VEL
LIN {X 0,Y 104.728,Z 976.392,A -85,B 0,C 180,E1 6020.672,E2 6020.672} C_VEL
LIN {X 0,Y 105.491,Z 975.05,A -85,B 0,C 180,E1 6010.639,E2 6010.639} C_VEL
LIN {X 0,Y 110.057,Z 971.67,A -85,B 0,C 180,E1 5998.216,E2 5998.216} C_VEL
LIN {X 0,Y 118.368,Z 966.73,A -85,B 0,C 180,E1 5987.502,E2 5987.502} C_VEL
LIN {X 0,Y 130.664,Z 959.654,A -85,B 0,C 180,E1 5978.003,E2 5978.003} C_VEL
LIN {X 0,Y 144.902,Z 951.134,A -85,B 0,C 180,E1 5970.704,E2 5970.704} C_VEL
LIN {X 0,Y 160.872,Z 940.889,A -85,B 0,C 180,E1 5964.87,E2 5964.87} C_VEL
LIN {X 0,Y 177.111,Z 929.472,A -85,B 0,C 180,E1 5960.449,E2 5960.449} C_VEL
LIN {X 0,Y 193.399,Z 916.704,A -85,B 0,C 180,E1 5957.002,E2 5957.002} C_VEL
LIN {X 0,Y 209.418,Z 902.576,A -85,B 0,C 180,E1 5954.284,E2 5954.284} C_VEL
LIN {X 0,Y 225.899,Z 886.158,A -85,B 0,C 180,E1 5952.027,E2 5952.027} C_VEL
LIN {X 0,Y 239.715,Z 870.505,A -85,B 0,C 180,E1 5950.44,E2 5950.44} C_VEL
LIN {X 0,Y 225.466,Z 885.707,A -85,B 0,C 180,E1 5948.585,E2 5948.585} C_VEL
LIN {X 0,Y 209.658,Z 900.368,A -85,B 0,C 180,E1 5946.172,E2 5946.172} C_VEL
LIN {X 0,Y 194.278,Z 912.861,A -85,B 0,C 180,E1 5943.354,E2 5943.354} C_VEL
LIN {X 0,Y 177.951,Z 924.48,A -85,B 0,C 180,E1 5939.675,E2 5939.675} C_VEL
LIN {X 0,Y 161.571,Z 934.571,A -85,B 0,C 180,E1 5934.977,E2 5934.977} C_VEL
LIN {X 0,Y 146.508,Z 942.685,A -85,B 0,C 180,E1 5929.286,E2 5929.286} C_VEL
LIN {X 0,Y 132.452,Z 949.332,A -85,B 0,C 180,E1 5921.969,E2 5921.969} C_VEL
LIN {X 0,Y 120.536,Z 954.223,A -85,B 0,C 180,E1 5912.854,E2 5912.854} C_VEL
LIN {X 0,Y 112.231,Z 957.149,A -85,B 0,C 180,E1 5902.711,E2 5902.711} C_VEL
LIN {X 0,Y 107.262,Z 958.415,A -85,B 0,C 180,E1 5891.423,E2 5891.423} C_VEL
LIN {X 0,Y 105.529,Z 958.139,A -85,B 0,C 180,E1 5881.392,E2 5881.392} C_VEL
LIN {X 0,Y 105.431,Z 956.989,A -85,B 0,C 180,E1 5872.28,E2 5872.28} C_VEL
LIN {X 0,Y 106.871,Z 954.557,A -85,B 0,C 180,E1 5862.414,E2 5862.414} C_VEL
LIN {X 0,Y 110.837,Z 950.547,A -85,B 0,C 180,E1 5852.057,E2 5852.057} C_VEL
LIN {X 0,Y 117.803,Z 944.625,A -85,B 0,C 180,E1 5842.185,E2 5842.185} C_VEL
LIN {X 0,Y 127.038,Z 937.096,A -85,B 0,C 180,E1 5833.787,E2 5833.787} C_VEL
LIN {X 0,Y 137.718,Z 928.204,A -85,B 0,C 180,E1 5826.909,E2 5826.909} C_VEL
LIN {X 0,Y 149.504,Z 917.808,A -85,B 0,C 180,E1 5821.207,E2 5821.207} C_VEL
LIN {X 0,Y 162.387,Z 905.399,A -85,B 0,C 180,E1 5816.34,E2 5816.34} C_VEL
LIN {X 0,Y 175.585,Z 891.167,A -85,B 0,C 180,E1 5812.33,E2 5812.33} C_VEL
LIN {X 0,Y 187.714,Z 876.43,A -85,B 0,C 180,E1 5809.263,E2 5809.263} C_VEL
LIN {X 0,Y 199.644,Z 860.007,A -85,B 0,C 180,E1 5806.669,E2 5806.669} C_VEL
LIN {X 0,Y 210.613,Z 842.702,A -85,B 0,C 180,E1 5804.587,E2 5804.587} C_VEL
LIN {X 0,Y 220.479,Z 824.677,A -85,B 0,C 180,E1 5802.907,E2 5802.907} C_VEL
LIN {X 0,Y 229.591,Z 804.84,A -85,B 0,C 180,E1 5801.486,E2 5801.486} C_VEL
LIN {X 0,Y 237.017,Z 785.119,A -85,B 0,C 180,E1 5800.403,E2 5800.403} C_VEL
LIN {X 0,Y 243.413,Z 763.812,A -85,B 0,C 180,E1 5799.52,E2 5799.52} C_VEL
LIN {X 0,Y 248.425,Z 741.265,A -85,B 0,C 180,E1 5798.844,E2 5798.844} C_VEL
LIN {X 0,Y 251.96,Z 717.009,A -85,B 0,C 180,E1 5798.338,E2 5798.338} C_VEL
LIN {X 0,Y 262.626,Z 626.833,A -85,B 0,C 180,E1 5796.708,E2 5796.708} C_VEL
LIN {X 0,Y 259.645,Z 620.355,A -85,B 0,C 180,E1 5793.312,E2 5793.312} C_VEL
LIN {X 0,Y 257.015,Z 614.6,A -85,B 0,C 180,E1 5789.481,E2 5789.481} C_VEL
LIN {X 0,Y 255.073,Z 610.66,A -85,B 0,C 180,E1 5785.627,E2 5785.627} C_VEL
LIN {X 0,Y 253.702,Z 607.588,A -85,B 0,C 180,E1 5780.918,E2 5780.918} C_VEL
LIN {X 0,Y 253.371,Z 607.151,A -85,B 0,C 180,E1 5775.332,E2 5775.332} C_VEL
LIN {X 0,Y 253.969,Z 608.012,A -85,B 0,C 180,E1 5771.814,E2 5771.814} C_VEL
LIN {X 0,Y 255.942,Z 611.988,A -85,B 0,C 180,E1 5766.506,E2 5766.506} C_VEL
LIN {X 0,Y 258.068,Z 616.295,A -85,B 0,C 180,E1 5762.888,E2 5762.888} C_VEL
LIN {X 0,Y 260.712,Z 621.61,A -85,B 0,C 180,E1 5759.451,E2 5759.451} C_VEL
LIN {X 0,Y 263.993,Z 628.476,A -85,B 0,C 180,E1 5755.983,E2 5755.983} C_VEL
LIN {X 0,Y 265.204,Z 631.446,A -85,B 0,C 180,E1 5754.8,E2 5754.8} C_VEL
LIN {X 0,Y 252.302,Z 743.825,A -85,B 0,C 180,E1 5752.722,E2 5752.722} C_VEL
LIN {X 0,Y 247.908,Z 766.085,A -85,B 0,C 180,E1 5752.181,E2 5752.181} C_VEL
LIN {X 0,Y 242.106,Z 786.942,A -85,B 0,C 180,E1 5751.552,E2 5751.552} C_VEL
LIN {X 0,Y 234.589,Z 808.152,A -85,B 0,C 180,E1 5750.68,E2 5750.68} C_VEL
LIN {X 0,Y 227.619,Z 824.521,A -85,B 0,C 180,E1 5749.793,E2 5749.793} C_VEL
LIN {X 0,Y 224.024,Z 831.36,A -85,B 0,C 180,E1 5749.592,E2 5749.592} C_VEL
LIN {X 0,Y 212.661,Z 848.046,A -85,B 0,C 180,E1 5749.792,E2 5749.792} C_VEL
LIN {X 0,Y 208.441,Z 854.386,A -85,B 0,C 180,E1 5749.482,E2 5749.482} C_VEL
LIN {X 0,Y 196.589,Z 872.493,A -85,B 0,C 180,E1 5747.58,E2 5747.58} C_VEL
LIN {X 0,Y 184.06,Z 889.191,A -85,B 0,C 180,E1 5745.245,E2 5745.245} C_VEL
LIN {X 0,Y 170.718,Z 904.9,A -85,B 0,C 180,E1 5742.27,E2 5742.27} C_VEL
LIN {X 0,Y 156.902,Z 919.228,A -85,B 0,C 180,E1 5738.511,E2 5738.511} C_VEL
LIN {X 0,Y 143.597,Z 931.704,A -85,B 0,C 180,E1 5733.941,E2 5733.941} C_VEL
LIN {X 0,Y 130.002,Z 943.448,A -85,B 0,C 180,E1 5727.797,E2 5727.797} C_VEL
LIN {X 0,Y 118.146,Z 953.162,A -85,B 0,C 180,E1 5720.379,E2 5720.379} C_VEL
LIN {X 0,Y 108.088,Z 961.333,A -85,B 0,C 180,E1 5711.068,E2 5711.068} C_VEL
LIN {X 0,Y 101.082,Z 967.588,A -85,B 0,C 180,E1 5700.309,E2 5700.309} C_VEL
LIN {X 0,Y 97.458,Z 972.119,A -85,B 0,C 180,E1 5688.557,E2 5688.557} C_VEL
LIN {X 0,Y 96.874,Z 974.596,A -85,B 0,C 180,E1 5678.321,E2 5678.321} C_VEL
LIN {X 0,Y 97.224,Z 975.568,A -85,B 0,C 180,E1 5671.191,E2 5671.191} C_VEL
LIN {X 0,Y 97.011,Z 975.812,A -85,B 0,C 180,E1 5665.283,E2 5665.283} C_VEL
LIN {X 0,Y 96.856,Z 975.302,A -85,B 0,C 180,E1 5655.669,E2 5655.669} C_VEL
LIN {X 0,Y 99.734,Z 973.037,A -85,B 0,C 180,E1 5642.553,E2 5642.553} C_VEL
LIN {X 0,Y 106.83,Z 969.129,A -85,B 0,C 180,E1 5630.49,E2 5630.49} C_VEL
LIN {X 0,Y 118.333,Z 963.153,A -85,B 0,C 180,E1 5619.763,E2 5619.763} C_VEL
LIN {X 0,Y 132.436,Z 955.622,A -85,B 0,C 180,E1 5611.468,E2 5611.468} C_VEL
LIN {X 0,Y 148.771,Z 946.266,A -85,B 0,C 180,E1 5604.888,E2 5604.888} C_VEL
LIN {X 0,Y 165.87,Z 935.479,A -85,B 0,C 180,E1 5599.914,E2 5599.914} C_VEL
LIN {X 0,Y 184.042,Z 922.616,A -85,B 0,C 180,E1 5595.96,E2 5595.96} C_VEL
LIN {X 0,Y 201.147,Z 908.816,A -85,B 0,C 180,E1 5593.059,E2 5593.059} C_VEL
LIN {X 0,Y 217.171,Z 894.223,A -85,B 0,C 180,E1 5590.88,E2 5590.88} C_VEL
LIN {X 0,Y 222.074,Z 889.442,A -85,B 0,C 180,E1 5590.285,E2 5590.285} C_VEL
LIN {X 0,Y 206.511,Z 903.122,A -85,B 0,C 180,E1 5588.071,E2 5588.071} C_VEL
LIN {X 0,Y 189.515,Z 916.119,A -85,B 0,C 180,E1 5585.145,E2 5585.145} C_VEL
LIN {X 0,Y 173.017,Z 927.084,A -85,B 0,C 180,E1 5581.612,E2 5581.612} C_VEL
LIN {X 0,Y 157.128,Z 936.348,A -85,B 0,C 180,E1 5577.283,E2 5577.283} C_VEL
LIN {X 0,Y 140.568,Z 944.648,A -85,B 0,C 180,E1 5571.31,E2 5571.31} C_VEL
LIN {X 0,Y 126.65,Z 950.616,A -85,B 0,C 180,E1 5564.354,E2 5564.354} C_VEL
LIN {X 0,Y 114.341,Z 955.175,A -85,B 0,C 180,E1 5555.397,E2 5555.397} C_VEL
LIN {X 0,Y 104.973,Z 958.048,A -85,B 0,C 180,E1 5544.476,E2 5544.476} C_VEL
LIN {X 0,Y 99.63,Z 959.194,A -85,B 0,C 180,E1 5532.892,E2 5532.892} C_VEL
LIN {X 0,Y 97.559,Z 958.811,A -85,B 0,C 180,E1 5521.497,E2 5521.497} C_VEL
LIN {X 0,Y 97.538,Z 957.464,A -85,B 0,C 180,E1 5511.012,E2 5511.012} C_VEL
LIN {X 0,Y 99.344,Z 954.849,A -85,B 0,C 180,E1 5500.425,E2 5500.425} C_VEL
LIN {X 0,Y 104.306,Z 950.342,A -85,B 0,C 180,E1 5488.89,E2 5488.89} C_VEL
LIN {X 0,Y 112.073,Z 944.334,A -85,B 0,C 180,E1 5478.93,E2 5478.93} C_VEL
LIN {X 0,Y 122.301,Z 936.575,A -85,B 0,C 180,E1 5470.406,E2 5470.406} C_VEL
LIN {X 0,Y 134.161,Z 927.119,A -85,B 0,C 180,E1 5463.424,E2 5463.424} C_VEL
LIN {X 0,Y 146.732,Z 916.332,A -85,B 0,C 180,E1 5457.884,E2 5457.884} C_VEL
LIN {X 0,Y 160.307,Z 903.484,A -85,B 0,C 180,E1 5453.21,E2 5453.21} C_VEL
LIN {X 0,Y 173.32,Z 889.723,A -85,B 0,C 180,E1 5449.597,E2 5449.597} C_VEL
LIN {X 0,Y 186.267,Z 874.228,A -85,B 0,C 180,E1 5446.593,E2 5446.593} C_VEL
LIN {X 0,Y 198.572,Z 857.263,A -85,B 0,C 180,E1 5444.143,E2 5444.143} C_VEL
LIN {X 0,Y 209.404,Z 840.031,A -85,B 0,C 180,E1 5442.254,E2 5442.254} C_VEL
LIN {X 0,Y 219.459,Z 821.408,A -85,B 0,C 180,E1 5440.675,E2 5440.675} C_VEL
LIN {X 0,Y 227.931,Z 802.885,A -85,B 0,C 180,E1 5439.455,E2 5439.455} C_VEL
LIN {X 0,Y 235.645,Z 782.279,A -85,B 0,C 180,E1 5438.412,E2 5438.412} C_VEL
LIN {X 0,Y 241.851,Z 761.018,A -85,B 0,C 180,E1 5437.613,E2 5437.613} C_VEL
LIN {X 0,Y 246.462,Z 739.614,A -85,B 0,C 180,E1 5437.025,E2 5437.025} C_VEL
LIN {X 0,Y 250.495,Z 710.647,A -85,B 0,C 180,E1 5436.47,E2 5436.47} C_VEL
LIN {X 0,Y 259.935,Z 631.945,A -85,B 0,C 180,E1 5435.076,E2 5435.076} C_VEL
LIN {X 0,Y 257.009,Z 625.399,A -85,B 0,C 180,E1 5431.29,E2 5431.29} C_VEL
LIN {X 0,Y 255.205,Z 621.474,A -85,B 0,C 180,E1 5428.299,E2 5428.299} C_VEL
LIN {X 0,Y 253.897,Z 618.523,A -85,B 0,C 180,E1 5425.42,E2 5425.42} C_VEL
LIN {X 0,Y 252.611,Z 615.512,A -85,B 0,C 180,E1 5420.869,E2 5420.869} C_VEL
LIN {X 0,Y 252.29,Z 615.074,A -85,B 0,C 180,E1 5415.399,E2 5415.399} C_VEL
LIN {X 0,Y 252.87,Z 616.005,A -85,B 0,C 180,E1 5411.866,E2 5411.866} C_VEL
LIN {X 0,Y 254.717,Z 619.848,A -85,B 0,C 180,E1 5406.764,E2 5406.764} C_VEL
LIN {X 0,Y 256.717,Z 624.053,A -85,B 0,C 180,E1 5403.238,E2 5403.238} C_VEL
LIN {X 0,Y 259.569,Z 629.944,A -85,B 0,C 180,E1 5399.449,E2 5399.449} C_VEL
LIN {X 0,Y 262.378,Z 636.24,A -85,B 0,C 180,E1 5396.388,E2 5396.388} C_VEL
LIN {X 0,Y 249.816,Z 743.341,A -85,B 0,C 180,E1 5394.464,E2 5394.464} C_VEL
LIN {X 0,Y 245.348,Z 765.633,A -85,B 0,C 180,E1 5393.945,E2 5393.945} C_VEL
LIN {X 0,Y 239.345,Z 786.864,A -85,B 0,C 180,E1 5393.34,E2 5393.34} C_VEL
LIN {X 0,Y 231.943,Z 807.42,A -85,B 0,C 180,E1 5392.542,E2 5392.542} C_VEL
LIN {X 0,Y 223.233,Z 827.267,A -85,B 0,C 180,E1 5391.501,E2 5391.501} C_VEL
LIN {X 0,Y 213.123,Z 846.509,A -85,B 0,C 180,E1 5390.155,E2 5390.155} C_VEL
LIN {X 0,Y 208.441,Z 854.386,A -85,B 0,C 180,E1 5389.482,E2 5389.482} C_VEL
LIN {X 0,Y 204.103,Z 860.736,A -85,B 0,C 180,E1 5389.135,E2 5389.135} C_VEL
LIN {X 0,Y 190.979,Z 876.012,A -85,B 0,C 180,E1 5389.012,E2 5389.012} C_VEL
LIN {X 0,Y 186.101,Z 881.797,A -85,B 0,C 180,E1 5388.529,E2 5388.529} C_VEL
LIN {X 0,Y 173.107,Z 897.494,A -85,B 0,C 180,E1 5386.037,E2 5386.037} C_VEL
LIN {X 0,Y 159.116,Z 912.44,A -85,B 0,C 180,E1 5382.794,E2 5382.794} C_VEL
LIN {X 0,Y 144.197,Z 926.519,A -85,B 0,C 180,E1 5378.44,E2 5378.44} C_VEL
LIN {X 0,Y 130.852,Z 937.865,A -85,B 0,C 180,E1 5373.4,E2 5373.4} C_VEL
LIN {X 0,Y 117.454,Z 948.433,A -85,B 0,C 180,E1 5366.554,E2 5366.554} C_VEL
LIN {X 0,Y 106.024,Z 957.096,A -85,B 0,C 180,E1 5358.175,E2 5358.175} C_VEL
LIN {X 0,Y 96.77,Z 964.215,A -85,B 0,C 180,E1 5347.576,E2 5347.576} C_VEL
LIN {X 0,Y 90.993,Z 969.525,A -85,B 0,C 180,E1 5335.389,E2 5335.389} C_VEL
LIN {X 0,Y 88.919,Z 973.023,A -85,B 0,C 180,E1 5323.01,E2 5323.01} C_VEL
LIN {X 0,Y 89.165,Z 974.591,A -85,B 0,C 180,E1 5313.228,E2 5313.228} C_VEL
LIN {X 0,Y 89.164,Z 975.064,A -85,B 0,C 180,E1 5307.443,E2 5307.443} C_VEL
LIN {X 0,Y 88.809,Z 974.809,A -85,B 0,C 180,E1 5297.002,E2 5297.002} C_VEL
LIN {X 0,Y 91.065,Z 973.193,A -85,B 0,C 180,E1 5283.964,E2 5283.964} C_VEL
LIN {X 0,Y 97.918,Z 969.757,A -85,B 0,C 180,E1 5270.739,E2 5270.739} C_VEL
LIN {X 0,Y 109.533,Z 964.426,A -85,B 0,C 180,E1 5259.132,E2 5259.132} C_VEL
LIN {X 0,Y 124.646,Z 957.239,A -85,B 0,C 180,E1 5249.987,E2 5249.987} C_VEL
LIN {X 0,Y 142.229,Z 948.025,A -85,B 0,C 180,E1 5242.965,E2 5242.965} C_VEL
LIN {X 0,Y 159.781,Z 937.694,A -85,B 0,C 180,E1 5238.009,E2 5238.009} C_VEL
LIN {X 0,Y 177.437,Z 926.052,A -85,B 0,C 180,E1 5234.288,E2 5234.288} C_VEL
LIN {X 0,Y 194.823,Z 913.14,A -85,B 0,C 180,E1 5231.45,E2 5231.45} C_VEL
LIN {X 0,Y 204.396,Z 905.248,A -85,B 0,C 180,E1 5230.142,E2 5230.142} C_VEL
LIN {X 0,Y 187.545,Z 917.604,A -85,B 0,C 180,E1 5227.486,E2 5227.486} C_VEL
LIN {X 0,Y 170.033,Z 928.708,A -85,B 0,C 180,E1 5224.045,E2 5224.045} C_VEL
LIN {X 0,Y 152.954,Z 938.05,A -85,B 0,C 180,E1 5219.727,E2 5219.727} C_VEL
LIN {X 0,Y 136.28,Z 945.913,A -85,B 0,C 180,E1 5214.103,E2 5214.103} C_VEL
LIN {X 0,Y 120.283,Z 952.244,A -85,B 0,C 180,E1 5206.497,E2 5206.497} C_VEL
LIN {X 0,Y 107.298,Z 956.471,A -85,B 0,C 180,E1 5197.266,E2 5197.266} C_VEL
LIN {X 0,Y 97.56,Z 959.011,A -85,B 0,C 180,E1 5186.088,E2 5186.088} C_VEL
LIN {X 0,Y 91.562,Z 959.944,A -85,B 0,C 180,E1 5172.973,E2 5172.973} C_VEL
LIN {X 0,Y 89.589,Z 959.481,A -85,B 0,C 180,E1 5161.621,E2 5161.621} C_VEL
LIN {X 0,Y 89.617,Z 957.994,A -85,B 0,C 180,E1 5150.22,E2 5150.22} C_VEL
LIN {X 0,Y 91.738,Z 955.315,A -85,B 0,C 180,E1 5138.763,E2 5138.763} C_VEL
LIN {X 0,Y 97.37,Z 950.676,A -85,B 0,C 180,E1 5126.455,E2 5126.455} C_VEL
LIN {X 0,Y 106.234,Z 944.332,A -85,B 0,C 180,E1 5115.801,E2 5115.801} C_VEL
LIN {X 0,Y 117.044,Z 936.666,A -85,B 0,C 180,E1 5107.382,E2 5107.382} C_VEL
LIN {X 0,Y 130.26,Z 926.667,A -85,B 0,C 180,E1 5100.158,E2 5100.158} C_VEL
LIN {X 0,Y 143.699,Z 915.486,A -85,B 0,C 180,E1 5094.715,E2 5094.715} C_VEL
LIN {X 0,Y 157.1,Z 903.106,A -85,B 0,C 180,E1 5090.464,E2 5090.464} C_VEL
LIN {X 0,Y 170.297,Z 889.454,A -85,B 0,C 180,E1 5087.065,E2 5087.065} C_VEL
LIN {X 0,Y 183.539,Z 873.916,A -85,B 0,C 180,E1 5084.212,E2 5084.212} C_VEL
LIN {X 0,Y 196.247,Z 856.719,A -85,B 0,C 180,E1 5081.87,E2 5081.87} C_VEL
LIN {X 0,Y 207.649,Z 838.717,A -85,B 0,C 180,E1 5080.032,E2 5080.032} C_VEL
LIN {X 0,Y 217.509,Z 820.49,A -85,B 0,C 180,E1 5078.598,E2 5078.598} C_VEL
LIN {X 0,Y 226.544,Z 800.607,A -85,B 0,C 180,E1 5077.392,E2 5077.392} C_VEL
LIN {X 0,Y 234.033,Z 780.429,A -85,B 0,C 180,E1 5076.455,E2 5076.455} C_VEL
LIN {X 0,Y 240.314,Z 758.784,A -85,B 0,C 180,E1 5075.705,E2 5075.705} C_VEL
LIN {X 0,Y 244.999,Z 736.264,A -85,B 0,C 180,E1 5075.147,E2 5075.147} C_VEL
LIN {X 0,Y 251.903,Z 682.505,A -85,B 0,C 180,E1 5074.221,E2 5074.221} C_VEL
LIN {X 0,Y 257.436,Z 637.386,A -85,B 0,C 180,E1 5073.472,E2 5073.472} C_VEL
LIN {X 0,Y 254.994,Z 631.764,A -85,B 0,C 180,E1 5069.932,E2 5069.932} C_VEL
LIN {X 0,Y 253.591,Z 628.569,A -85,B 0,C 180,E1 5067.345,E2 5067.345} C_VEL
LIN {X 0,Y 252.553,Z 626.105,A -85,B 0,C 180,E1 5064.813,E2 5064.813} C_VEL
LIN {X 0,Y 251.454,Z 623.355,A -85,B 0,C 180,E1 5060.483,E2 5060.483} C_VEL
LIN {X 0,Y 251.26,Z 623.045,A -85,B 0,C 180,E1 5054.991,E2 5054.991} C_VEL
LIN {X 0,Y 251.725,Z 623.821,A -85,B 0,C 180,E1 5052.153,E2 5052.153} C_VEL
LIN {X 0,Y 253.439,Z 627.571,A -85,B 0,C 180,E1 5047.139,E2 5047.139} C_VEL
LIN {X 0,Y 255.286,Z 631.642,A -85,B 0,C 180,E1 5043.706,E2 5043.706} C_VEL
LIN {X 0,Y 257.977,Z 637.44,A -85,B 0,C 180,E1 5039.971,E2 5039.971} C_VEL
LIN {X 0,Y 259.635,Z 641.45,A -85,B 0,C 180,E1 5037.989,E2 5037.989} C_VEL
LIN {X 0,Y 247.452,Z 743.133,A -85,B 0,C 180,E1 5036.228,E2 5036.228} C_VEL
LIN {X 0,Y 242.893,Z 765.508,A -85,B 0,C 180,E1 5035.734,E2 5035.734} C_VEL
LIN {X 0,Y 236.822,Z 786.64,A -85,B 0,C 180,E1 5035.169,E2 5035.169} C_VEL
LIN {X 0,Y 229.076,Z 807.743,A -85,B 0,C 180,E1 5034.397,E2 5034.397} C_VEL
LIN {X 0,Y 220.166,Z 827.587,A -85,B 0,C 180,E1 5033.409,E2 5033.409} C_VEL
LIN {X 0,Y 209.955,Z 846.656,A -85,B 0,C 180,E1 5032.145,E2 5032.145} C_VEL
LIN {X 0,Y 198.677,Z 864.51,A -85,B 0,C 180,E1 5030.561,E2 5030.561} C_VEL
LIN {X 0,Y 186.101,Z 881.797,A -85,B 0,C 180,E1 5028.529,E2 5028.529} C_VEL
LIN {X 0,Y 181.125,Z 887.53,A -85,B 0,C 180,E1 5027.996,E2 5027.996} C_VEL
LIN {X 0,Y 166.41,Z 901.162,A -85,B 0,C 180,E1 5027.419,E2 5027.419} C_VEL
LIN {X 0,Y 160.986,Z 906.269,A -85,B 0,C 180,E1 5026.671,E2 5026.671} C_VEL
LIN {X 0,Y 147.2,Z 919.591,A -85,B 0,C 180,E1 5023.308,E2 5023.308} C_VEL
LIN {X 0,Y 132.112,Z 932.491,A -85,B 0,C 180,E1 5018.595,E2 5018.595} C_VEL
LIN {X 0,Y 118.113,Z 943.312,A -85,B 0,C 180,E1 5012.749,E2 5012.749} C_VEL
LIN {X 0,Y 104.316,Z 953.223,A -85,B 0,C 180,E1 5004.577,E2 5004.577} C_VEL
LIN {X 0,Y 93.557,Z 960.795,A -85,B 0,C 180,E1 4994.874,E2 4994.874} C_VEL
LIN {X 0,Y 85.509,Z 966.852,A -85,B 0,C 180,E1 4982.555,E2 4982.555} C_VEL
LIN {X 0,Y 81.443,Z 971.13,A -85,B 0,C 180,E1 4968.63,E2 4968.63} C_VEL
LIN {X 0,Y 81.01,Z 973.46,A -85,B 0,C 180,E1 4956.393,E2 4956.393} C_VEL
LIN {X 0,Y 81.3,Z 974.138,A -85,B 0,C 180,E1 4949.31,E2 4949.31} C_VEL
LIN {X 0,Y 80.821,Z 974.267,A -85,B 0,C 180,E1 4940.761,E2 4940.761} C_VEL
LIN {X 0,Y 82.262,Z 973.252,A -85,B 0,C 180,E1 4926.37,E2 4926.37} C_VEL
LIN {X 0,Y 88.598,Z 970.469,A -85,B 0,C 180,E1 4911.652,E2 4911.652} C_VEL
LIN {X 0,Y 99.862,Z 965.871,A -85,B 0,C 180,E1 4899.106,E2 4899.106} C_VEL
LIN {X 0,Y 115.593,Z 959.196,A -85,B 0,C 180,E1 4888.971,E2 4888.971} C_VEL
LIN {X 0,Y 132.559,Z 951.269,A -85,B 0,C 180,E1 4881.941,E2 4881.941} C_VEL
LIN {X 0,Y 151.793,Z 941.091,A -85,B 0,C 180,E1 4876.453,E2 4876.453} C_VEL
LIN {X 0,Y 170.997,Z 929.399,A -85,B 0,C 180,E1 4872.491,E2 4872.491} C_VEL
LIN {X 0,Y 186.585,Z 918.656,A -85,B 0,C 180,E1 4869.978,E2 4869.978} C_VEL
LIN {X 0,Y 168.618,Z 929.655,A -85,B 0,C 180,E1 4866.81,E2 4866.81} C_VEL
LIN {X 0,Y 150.104,Z 939.32,A -85,B 0,C 180,E1 4862.57,E2 4862.57} C_VEL
LIN {X 0,Y 133.098,Z 946.865,A -85,B 0,C 180,E1 4857.346,E2 4857.346} C_VEL
LIN {X 0,Y 116.356,Z 953.055,A -85,B 0,C 180,E1 4850.102,E2 4850.102} C_VEL
LIN {X 0,Y 101.761,Z 957.389,A -85,B 0,C 180,E1 4840.565,E2 4840.565} C_VEL
LIN {X 0,Y 90.833,Z 959.859,A -85,B 0,C 180,E1 4828.843,E2 4828.843} C_VEL
LIN {X 0,Y 83.846,Z 960.697,A -85,B 0,C 180,E1 4814.314,E2 4814.314} C_VEL
LIN {X 0,Y 81.569,Z 960.096,A -85,B 0,C 180,E1 4800.967,E2 4800.967} C_VEL
LIN {X 0,Y 81.789,Z 958.378,A -85,B 0,C 180,E1 4788.516,E2 4788.516} C_VEL
LIN {X 0,Y 84.689,Z 955.396,A -85,B 0,C 180,E1 4775.405,E2 4775.405} C_VEL
LIN {X 0,Y 91.477,Z 950.441,A -85,B 0,C 180,E1 4762.45,E2 4762.45} C_VEL
LIN {X 0,Y 100.979,Z 944.143,A -85,B 0,C 180,E1 4752.112,E2 4752.112} C_VEL
LIN {X 0,Y 113.479,Z 935.726,A -85,B 0,C 180,E1 4743.286,E2 4743.286} C_VEL
LIN {X 0,Y 126.839,Z 926.05,A -85,B 0,C 180,E1 4736.679,E2 4736.679} C_VEL
LIN {X 0,Y 141.119,Z 914.592,A -85,B 0,C 180,E1 4731.418,E2 4731.418} C_VEL
LIN {X 0,Y 155.106,Z 901.89,A -85,B 0,C 180,E1 4727.392,E2 4727.392} C_VEL
LIN {X 0,Y 168.77,Z 887.879,A -85,B 0,C 180,E1 4724.197,E2 4724.197} C_VEL
LIN {X 0,Y 182.59,Z 871.692,A -85,B 0,C 180,E1 4721.499,E2 4721.499} C_VEL
LIN {X 0,Y 194.876,Z 855.118,A -85,B 0,C 180,E1 4719.443,E2 4719.443} C_VEL
LIN {X 0,Y 206.667,Z 836.601,A -85,B 0,C 180,E1 4717.712,E2 4717.712} C_VEL
LIN {X 0,Y 217.184,Z 816.944,A -85,B 0,C 180,E1 4716.32,E2 4716.32} C_VEL
LIN {X 0,Y 225.813,Z 797.448,A -85,B 0,C 180,E1 4715.263,E2 4715.263} C_VEL
LIN {X 0,Y 233.292,Z 776.607,A -85,B 0,C 180,E1 4714.402,E2 4714.402} C_VEL
LIN {X 0,Y 239.444,Z 754.298,A -85,B 0,C 180,E1 4713.72,E2 4713.72} C_VEL
LIN {X 0,Y 243.723,Z 732.456,A -85,B 0,C 180,E1 4713.247,E2 4713.247} C_VEL
LIN {X 0,Y 255.015,Z 642.855,A -85,B 0,C 180,E1 4711.761,E2 4711.761} C_VEL
LIN {X 0,Y 252.784,Z 637.319,A -85,B 0,C 180,E1 4707.952,E2 4707.952} C_VEL
LIN {X 0,Y 251.407,Z 634.023,A -85,B 0,C 180,E1 4704.683,E2 4704.683} C_VEL
LIN {X 0,Y 250.348,Z 631.256,A -85,B 0,C 180,E1 4700.333,E2 4700.333} C_VEL
LIN {X 0,Y 250.217,Z 631.01,A -85,B 0,C 180,E1 4694.743,E2 4694.743} C_VEL
LIN {X 0,Y 250.629,Z 631.825,A -85,B 0,C 180,E1 4692.19,E2 4692.19} C_VEL
LIN {X 0,Y 252.211,Z 635.426,A -85,B 0,C 180,E1 4687.403,E2 4687.403} C_VEL
LIN {X 0,Y 253.936,Z 639.394,A -85,B 0,C 180,E1 4684.065,E2 4684.065} C_VEL
LIN {X 0,Y 256.473,Z 645.137,A -85,B 0,C 180,E1 4680.392,E2 4680.392} C_VEL
LIN {X 0,Y 257.064,Z 646.811,A -85,B 0,C 180,E1 4679.625,E2 4679.625} C_VEL
LIN {X 0,Y 245.312,Z 742.788,A -85,B 0,C 180,E1 4678.025,E2 4678.025} C_VEL
LIN {X 0,Y 240.683,Z 765.156,A -85,B 0,C 180,E1 4677.558,E2 4677.558} C_VEL
LIN {X 0,Y 234.545,Z 786.24,A -85,B 0,C 180,E1 4677.035,E2 4677.035} C_VEL
LIN {X 0,Y 226.944,Z 806.738,A -85,B 0,C 180,E1 4676.345,E2 4676.345} C_VEL
LIN {X 0,Y 218.191,Z 826.119,A -85,B 0,C 180,E1 4675.46,E2 4675.46} C_VEL
LIN {X 0,Y 207.529,Z 845.777,A -85,B 0,C 180,E1 4674.253,E2 4674.253} C_VEL
LIN {X 0,Y 196.045,Z 863.721,A -85,B 0,C 180,E1 4672.772,E2 4672.772} C_VEL
LIN {X 0,Y 183.308,Z 880.951,A -85,B 0,C 180,E1 4670.879,E2 4670.879} C_VEL
LIN {X 0,Y 170.355,Z 896.328,A -85,B 0,C 180,E1 4668.598,E2 4668.598} C_VEL
LIN {X 0,Y 160.986,Z 906.269,A -85,B 0,C 180,E1 4666.671,E2 4666.671} C_VEL
LIN {X 0,Y 155.471,Z 911.32,A -85,B 0,C 180,E1 4665.845,E2 4665.845} C_VEL
LIN {X 0,Y 139.467,Z 923.026,A -85,B 0,C 180,E1 4664.579,E2 4664.579} C_VEL
LIN {X 0,Y 133.634,Z 927.346,A -85,B 0,C 180,E1 4663.421,E2 4663.421} C_VEL
LIN {X 0,Y 118.492,Z 939.014,A -85,B 0,C 180,E1 4658.179,E2 4658.179} C_VEL
LIN {X 0,Y 104.342,Z 948.825,A -85,B 0,C 180,E1 4651.373,E2 4651.373} C_VEL
LIN {X 0,Y 91.3,Z 957.324,A -85,B 0,C 180,E1 4642.065,E2 4642.065} C_VEL
LIN {X 0,Y 80.993,Z 964.12,A -85,B 0,C 180,E1 4629.955,E2 4629.955} C_VEL
LIN {X 0,Y 74.935,Z 968.861,A -85,B 0,C 180,E1 4616.142,E2 4616.142} C_VEL
LIN {X 0,Y 72.934,Z 972.007,A -85,B 0,C 180,E1 4601.082,E2 4601.082} C_VEL
LIN {X 0,Y 73.308,Z 973.172,A -85,B 0,C 180,E1 4591.58,E2 4591.58} C_VEL
LIN {X 0,Y 73.025,Z 973.554,A -85,B 0,C 180,E1 4584.517,E2 4584.517} C_VEL
LIN {X 0,Y 73.462,Z 973.096,A -85,B 0,C 180,E1 4570.125,E2 4570.125} C_VEL
LIN {X 0,Y 78.543,Z 971.208,A -85,B 0,C 180,E1 4554.176,E2 4554.176} C_VEL
LIN {X 0,Y 89.889,Z 967.209,A -85,B 0,C 180,E1 4539.345,E2 4539.345} C_VEL
LIN {X 0,Y 104.854,Z 961.64,A -85,B 0,C 180,E1 4528.711,E2 4528.711} C_VEL
